	//M_EXECUTE VARIABLES //
		TP_READ						: LTP;  //Tempo de cadencement FB Modbus
		RTrig						: R_Trig; //Front montant sur TP_READ.Q
		ReadBusy					: BOOL;	//FB Modbus en busy



	
END_VAR

METHOD M_Execute
//////////////////
//  Method Calls 
/////////////////

VAR 
	// Method local variables (reinitialized at each cycle) 
	
	SppNum: UINT;
MesDataExd.MesData.NV: INT;
	SetTempSlope: REAL;
END_VAR

FOR KK_ModbusRead:=1 TO 2 DO
	AX_Error[KK_ModbusRead] 			:= Emul_MesModbusReadAlarm[KK_ModbusRead] ;
	
END_FOR

// INV 
SppNum:= SEL(ParamUnitID>11 ,1 , 2) ; 
		
			AX_PTR[SppNum].A1_INV_Smartlogger.Emul_RS(SET1:= IN_CmdStop, RESET:=IN_CmdStart ) ; 
			IF Emul_AlarmINV  THEN 
			MesDataExd.MesData.MesIDState :=16#0300 ;

			ELSIF AX_PTR[SppNum].A1_INV_Smartlogger.Emul_RS.Q1 THEN 
			MesDataExd.MesData.MesIDState:=16#0304 ;

			ELSIF MesP_INVmppt=0 THEN 
			MesDataExd.MesData.MesIDState:=16#A000 ;
	
			ELSIF IN_SetptPlimit < ParamPn THEN 
			MesDataExd.MesData.MesIDState:=16#0202 ;

			ELSIF AX_PTR[SppNum].A1_INV_Smartlogger.Emul_ComError THEN 
			MesDataExd.MesData.MesIDState:=16#B000 ;

			ELSE
			MesDataExd.MesData.MesIDState:=16#0200 ;

			END_IF	
	// Pas de pente dans les onduleurs . 		
//			Emul_Smooth(Setpoint:= AX_SPP[SppNum].A1_SmartLogger.SetptPlimit/AX_SPP[SppNum].A1_SmartLogger.ParamNbINV , Slope :=5,DeadBand:=2,Range:= ParamPnom,CycleTime:=CstCycleTime_G,InitialValue:=0, Reset:=(A1_HPP.CalState =9) OR Emul_AlarmINV OR NOT(AX_SPP[SppNum].A1_TGBT.MesDataExd.MesData.MesMainCB), OutValue=> SetTempSlope ) ;
			SetTempSlope :=SEL( MesDataExd.MesData.MesAlarmCom ,  AX_PTR[SppNum].A1_INV_Smartlogger.IN_SetptPlimit/AX_PTR[SppNum].A1_INV_Smartlogger.ParamNbINV , AX_PTR[SppNum].A1_INV_Smartlogger.ParamPnomINV )  ; 

		MesDataExd.MesData.MesP 			:=SEL((A1_PP.MesState =9) OR AX_PTR[SppNum].A1_INV_Smartlogger.Emul_AlarmINV OR NOT(AX_PTR[SppNum].A1_MainMVCB_PTR.MesDataExd.MesData.MesClosed) , MIN(SetTempSlope , MesP_INVmppt),  0)  ; 
		MesDataExd.MesData.MesQ 			:= AX_PTR[SppNum].A1_INV_Smartlogger.IN_SetptQlimit/AX_PTR[SppNum].A1_INV_Smartlogger.ParamNbINV  ; 
		MesDataExd.MesData.MesPdc 			:= MesDataExd.MesData.MesP/AX_PTR[SppNum].A1_INV_Smartlogger.MesDataExd.MesData.MesEff; 
		MesDataExd.MesData.MesIdc 			:= MesDataExd.MesData.MesPdc 	MesDataExd.MesData.MesUdc; 



MesDataExd.MesData.MesU 			:= AX_PTR[SppNum].A1_INV_Smartlogger.MesDataExd.MesData.MesU12 ; 
MesDataExd.MesData.MesV			    := MesDataExd.MesData.MesU/SQRT(3)*2 ; 
MesDataExd.MesData.MesI			    := SEL.MesDataExd.MesData.MesU = 0 , MesDataExd.MesData.MesP*1000 MesDataExd.MesData.MesU /SQRT(3) ,0 ) ; 
MesDataExd.MesData.MesFreq			:=  A1_SUBMV.A1_PM.MesDataExd.MesData.Mesfreq; 
MesDataExd.MesData.MesS			    := SQRT.MesDataExd.MesData.MesP.MesDataExd.MesData.MesP.MesDataExd.MesData.MesQ.MesDataExd.MesData.MesQ) ; 

MesDataExd.MesData.MesCosPhi			:=  0.95  ; 
MesDataExd.MesData.MesTemp			:= 32 ;  


// Other Variables
//MesDataExd.MesData.MesInsuResistor			:= 1220 ; 	

// Properties update. 
MesDataExd.MesData.MesAlarmCom	:= MesDataExd.MesData.MesIDState = 16#B000 ; 

//MesDataExd.MesData.MesAlm1		:= MesDataExd.MesData.MesIDState = 16#0300 ;
MesDataExd.MesData.ParamPn		:= 60  ; 

//MesDataExd.MesData.CalCurtailing	:= MesDataExd.MesData.MesStatus = 16#0201 OR MesDataExd.MesData.MesStatus = 16#0202; 
	

MesDataExd.MesData.MesUdc			:= 200 ;
MesDataExd.MesData.MesInsuResistor 	:= 150 ;
//MesDataExd.MesData.MesPF			:=0.97 ; 


//INV Exd
MesDataExd.MesEDay			:= 1000 ; 
MesDataExd.MesETot			:=  1100; 
MesDataExd.MesI1			:= MesDataExd.MesData.MesI; 
MesDataExd.MesI2			:= MesDataExd.MesData.MesI; 
MesDataExd.MesI3			:= MesDataExd.MesData.MesI; 
MesDataExd.MesU12			:=  AX_PTR[SppNum].A1_INV_Smartlogger.MesDataExd.MesData.MesU12; 
MesDataExd.MesU23			:=   AX_PTR[SppNum].A1_INV_Smartlogger.MesDataExd.MesData.MesU23; 
MesDataExd.MesU31			:=   AX_PTR[SppNum].A1_INV_Smartlogger.MesDataExd.MesData.MesU31; 
MesDataExd.MesV1			:= MesDataExd.MesData.MesV; 
MesDataExd.MesV2			:= MesDataExd.MesData.MesV;  
MesDataExd.MesV3			:= MesDataExd.MesData.MesV; 


// Properties update.
MesDataExd.MesData.MesI := MesDataExd.MesData.MesI1 + MesDataExd.MesData.MesI2 + MesDataExd.MesData.MesI3)/3;
MesDataExd.MesData.MesV := MesDataExd.MesData.MesV1 + MesDataExd.MesData.MesV2 + MesDataExd.MesData.MesV3)/3;
MesDataExd.MesData.MesS := SQRT.MesDataExd.MesData.MesP.MesDataExd.MesData.MesP + MesDataExd.MesData.MesQ.MesDataExd.MesData.MesQ);

MesDataExd.MesData.MesCurtl := MesDataExd.MesData.MesIDState=16#0202 OR MesDataExd.MesData.MesIDState=16#0203 ; 
//MesDataExd.MesData.ParamPnom := ParamPnom ;
END_METHOD

END_FUNCTION_BLOCK

// ---- 01_Equipement_Library/IPC/FB_IPC.TcPOU
FUNCTION_BLOCK FB_IPC

VAR_INPUT PERSISTENT 
	ParamTempoRestart		: TIME 	:= T#30S ;	(*  (s)Tempo to wait before resupplying the IPC*)
	
END_VAR
      	
VAR_INPUT           	
	Heure_Local     		: TIMESTRUCT;
	IN_CmdRestart 			: BOOL;	
	IN_CmdReset_L			: BOOL;			// (NA) External Reset Command
	
END_VAR     

VAR_OUTPUT
	//Child objects
	OUT_CmdOpen_IO			: BOOL;	
END_VAR        	
      	
VAR                 	
	bInit					: BOOL := TRUE;	// Booleen d'initialisation
		
	TP_Restart				: TP;
	// State Mananger //
	MesState				: BYTE; 		// Cal  : state
	
	// M_Evaluate //	
	MesData			: IPC;
	
END_VAR

METHOD M_Execute : BOOL
VAR_INPUT
END_VAR
END_METHOD

END_FUNCTION_BLOCK

// ---- 01_Equipement_Library/Operation Meter/FB_PM_520_230.TcPOU
FUNCTION_BLOCK FB_PM_520_230 EXTENDS FB_PM_Base
//////////////////
// Measurement Solution based on Digiware, but access through PMS Socomec
//////////////////
VAR CONSTANT
	// Characteristics of the object (Same for all instances)
			
END_VAR

VAR_INPUT PERSISTENT
	// Parameters of the Object (instance specific) 
	ParamUnitID					: BYTE 		:= 1 ;								// (NA)unit ID
	ParamInInterfaceSub			: BOOL := TRUE; // Serial interface RS422/RS485 TYPE (0:EL6021,1:SUB9)			
END_VAR

VAR_OUTPUT
	//Child objects
	
END_VAR
VAR
	//M_ALARMMANAGEMENT VARIABLES//
	                                                    								
                                                        								

	//M_READ VARIABLES//
		ModbusRTU					: FB_ModbusRTU;				// (NA) FB for Modbus Reading
				// (NA) Start address of the read
		//MesDataExd				: PM520;								// (NA) Structure of the PM3250
		
		ObjectCom					: INT;									// (NA) Sequence index
									
		Busy						: BOOL;
		StepRead					: UINT;									// (NA) Step for reading 2 blocks of registers
		AX_TrigRead					: ARRAY[1..1] OF R_trig;
		MbStruct					: ARRAY[1..1] OF Struct_InputRTU;	
		MesBlock					: ARRAY[1..1] OF ARRAY[1..120] OF WORD;	
		AX_Addr						: ARRAY[1..1] OF UINT 	:= [19000];
		AX_Qty						: ARRAY[1..1] OF UINT	:= [86];
		AX_UnitId					: ARRAY[1..1] OF BYTE	:= [1];
		AX_Function					: ARRAY[1..1] OF UINT	:= [4];	
		AX_Priority					: ARRAY[1..1] OF UINT	:= [1];
		KK							: INT;
		ComError 					: BOOL;
	//M_INIT VARIABLES //
		OutFBCompleteted			: BOOL;
	// M_EXECUTE VARIABLES //
		
                              

 
END_VAR

METHOD M_Execute
//////////////////
//  Method Calls 
/////////////////
VAR 

	
END_VAR
END_METHOD

END_FUNCTION_BLOCK

// ---- 01_Equipement_Library/Operation Meter/FB_PM_Base.TcPOU
FUNCTION_BLOCK FB_PM_Base 
//////////////////
// Measurement Solution. Base FB
//////////////////
VAR_INPUT PERSISTENT
	// Parameters of the Object (instance specific) 
	ParamTempoComAlarm			: TIME 			:= T#10S ; 						// (s) Config : Tempo to detect LOC Alarm
	ParamClockReadTime 			: TIME 			:= TIME#200MS;	  				// (ms) Read Modbus Frequency.  
	ParamTimeout				: TIME  		:= T#2S ;			  			// (s) Timeout for modbus reading
	
	
END_VAR

VAR_INPUT
	//Child objects
	IN_CmdToggleRead				: BOOL ; 
	IN_CmdReset_L					: BOOL ;	// (NA) External Reset Command

END_VAR
VAR
	//M_ALARMMANAGEMENT VARIABLES//
		TON_ComAlarm				: TON ; 												// Tempo before detecting loss of communication. 
	    TON_ComWarning				: TON ; 												// Tempo before detecting loss of one frame.                                               								
                                            								
												//(NA) [P,H] Communication Error with D50 Digiware (all chain ) 
		MesWarningCom				: BOOL ; 												// True if bad communication .

	//M_READ VARIABLES//
//	MesDataExd				AT %Q*: PM ; 
		ClockRead					AT %Q*: BOOL ; 												// Clock Read

	//M_INIT VARIABLES //
		bInit						: BOOL 				:= TRUE ; 							// (NA) Initialize object parameters at first cycle 
		
	// M_EXECUTE VARIABLES //
		TP1							: TP ; 												// (NA) Tempo to define Modbus Reading Frequency  
		
		//MesCP_Read					: BOOL;													// (NA) Permanent conditions to activate method
        Trig_Cmd_Read				: R_TRIG;                       
	// EMULATOR //                      
		
 
END_VAR

METHOD M_Execute
//////////////////
//  Method Calls 
/////////////////
VAR 
	// Method local variables (reinitialized at each cycle) 
	// EMULATOR

	
END_VAR
END_METHOD

END_FUNCTION_BLOCK

// ---- 01_Equipement_Library/Operation Meter/FB_PM_A40.TcPOU
FUNCTION_BLOCK FB_PM_A40 EXTENDS FB_PM_Base
//////////////////
// Measurement Solution based on Digiware, but access through PMS Socomec
//////////////////

VAR_INPUT PERSISTENT
	// Parameters of the Object (instance specific) 
	ParamUnitID					: BYTE := 22; 							// (NA) All unit ID For the Device (I35 + 1 U20)                                                                    			
	                                                                            			
	ParamIPAddress			   	: STRING := '192.168.20.15'; 								// (NA) IP Adress of D50 .
	ParamTCPPort				: UINT := 502;		// Modbus TCP Port


END_VAR

VAR_OUTPUT
	//Child objects
	
END_VAR
VAR
	//M_ALARMMANAGEMENT VARIABLES//
		
	//M_READ VARIABLES//
		FB_ModbusRead_I1			: ARRAY[1..2] OF  FB_ModbusRead ; 			// (NA) FB for Modbus Reading
	                                                                                    	
		MesBlock1_Temp 				: ARRAY[1..2] 	OF ARRAY[0..124] OF WORD;		//(NA) Temporary Block with multiple modbus reading (U30 + I35)
		MesModbusReadAlarm 		  	: ARRAY[1..2] OF BOOL ; 						// (NA) Modbus Read Alarm for communication 
		
		
		MesModbusAlarmCode			: ARRAY[1..2] OF UDINT;						// (NA) Modbus Read Alarm Code	
		
	//M_INIT VARIABLES //
		
	// M_EXECUTE VARIABLES //
		   	MesDataExd AT %Q*			: PM_Standard ;               


 
END_VAR

METHOD M_Execute
//////////////////
//  Method Calls 
/////////////////
VAR 
MesDataExd.MesData.dl 		: PDL_Exd;
	MesStateCB 		: BOOL;
MesDataExd.MesData.ull		: PM;
	
	KK: INT;
END_VAR
 MesDataExd.MesData.dl := A1_SUBMV.MesDataExd.MesData.

MesStateCB := A1_SUBMV.A1_MainMVCB.MesDataExd.MesData.MesClosed ; 
MesData.MesP := 0 ;
MesData.MesQ := 0 ; 


IF MesStateCB THEN
MesDataExd.MesData.MesU 	:= 230;
MesDataExd.MesData.MesU12 	:= 230;
MesDataExd.MesData.MesU23 	:= 230;
MesDataExd.MesData.MesU31 	:= 230;
MesDataExd.MesData.MesV 	:= A1_PP.MesDataExd.MesData.MesU/SQRT(3);
MesDataExd.MesData.MesV1 	:= A1_PP.MesDataExd.MesData.MesU/SQRT(3);
MesDataExd.MesData.MesV2 	:= A1_PP.MesDataExd.MesData.MesU/SQRT(3);
MesDataExd.MesData.MesV3 	:= A1_PP.MesDataExd.MesData.MesU/SQRT(3);
MesDataExd.MesData.MesFreq := A1_PP.MesDataExd.MesData.MesFreq;
	
	

MesDataExd.MesData.MesP 	:= 120  ;
MesDataExd.MesData.MesQ 	:= -20 ;
	
	
MesDataExd.MesData.MesP1 	:= MesDataExd.MesData.MesP ;
MesDataExd.MesData.MesP2 	:= 0 ;
MesDataExd.MesData.MesP3 	:= 0 ;

MesDataExd.MesData.MesQ1 	:= MesDataExd.MesData.MesQ;
MesDataExd.MesData.MesQ2 	:= 0;
MesDataExd.MesData.MesQ3 	:= 0;
MesDataExd.MesData.MesS := SQRT( MesDataExd.MesData.MesP * MesDataExd.MesData.MesP + MesDataExd.MesData.MesQ.MesDataExd.MesData.MesQ ) ; 
	
MesDataExd.MesData.MesI 	:= MesDataExd.MesData.MesS/(SQRT(3)*A1_PP.MesDataExd.MesData.MesU);
MesDataExd.MesData.MesI1 	:= MesDataExd.MesData.MesS/(SQRT(3)*A1_PP.MesDataExd.MesData.MesU);

ELSE 
MesDataExd.MesData.:= MesDataExd.MesData.ull;
END_IF

IF MesDataExd.MesData.MesP > 0 THEN
MesDataExd.MesData.MesE_AcDel := MesDataExd.MesData.MesE_AcDel + MesDataExd.MesData.MesP*ParamCycleTime_Emul/3600000	;
END_IF
IF MesDataExd.MesData.MesP < 0 THEN
MesDataExd.MesData.MesE_AcRec := MesDataExd.MesData.MesE_AcRec -.MesDataExd.MesData.MesP*ParamCycleTime_Emul/3600000	;
END_IF
IF MesDataExd.MesData.MesQ > 0 THEN
MesDataExd.MesData.MesE_ReacDel := MesDataExd.MesData.MesE_ReacDel + MesDataExd.MesData.MesQ*ParamCycleTime_Emul/3600000	;
END_IF
IF MesDataExd.MesData.MesQ < 0 THEN
MesDataExd.MesData.MesE_ReacRec := MesDataExd.MesData.MesE_ReacRec -.MesDataExd.MesData.MesQ*ParamCycleTime_Emul/3600000	;
END_IF

MesDataNull.MesE_ReacRec := MesDataExd.MesData.MesE_ReacRec;	
MesDataNull.MesE_ReacDel := MesDataExd.MesData.MesE_ReacDel;	
MesDataNull.MesE_AcRec := MesDataExd.MesData.MesE_AcRec;		
MesDataNull.MesE_AcDel := MesDataExd.MesData.MesE_AcDel;
END_METHOD

END_FUNCTION_BLOCK

// ---- 01_Equipement_Library/Operation Meter/FB_PM_ION7650.TcPOU
FUNCTION_BLOCK FB_PM_ION7650 EXTENDS FB_PM_Base
//////////////////
// Measurement Solution based on Digiware, but access through PMS Socomec
//////////////////
VAR CONSTANT
	// Characteristics of the object (Same for all instances)
			
END_VAR

VAR_INPUT PERSISTENT
	// Parameters of the Object (instance specific) 
	ParamUnitID					: BYTE 		:= 1 ;								// (NA)unit ID
//	ParamInInterfaceSub			: BOOL := TRUE; // Serial interface RS422/RS485 TYPE (0:EL6021,1:SUB9)
	ParamIPAdress		   		: STRING 	:= '192.168.20.15'; 				// (NA) IP Adress of ION7650 .
	ParamTcpPort				: UINT 		:= 502;					
	
END_VAR

VAR_OUTPUT
	//Child objects
	
END_VAR
VAR
	//M_ALARMMANAGEMENT VARIABLES//
	                                                    								                                          								

	//M_READ VARIABLES//
		FB_ModbusRead				: FB_ModbusRTU ;					// (NA) FB for Modbus Reading
		InputStructRead 			: ARRAY[1..1] OF  Struct_InputRTU;
		
		AX_Quantity					: ARRAY[1..1] OF WORD;					// (NA) Quantity of blocks to read
		AX_Address					: ARRAY[1..1] OF WORD;					// (NA) Start address of the read
		MesBlock_Temp 				: ARRAY[1..1] OF ARRAY[1..125] OF WORD;	// (NA) Temporary Block with multiple modbus reading (U30 + I35)
		Busy						: BOOL;
		OutErrorMbRead				: ARRAY[1..1] OF BOOL;
		
		RTrigI						: R_TRIG;
	//M_INIT VARIABLES //
		OutFBCompleteted			: BOOL;
	// M_EXECUTE VARIABLES //
 
	MesDataExd AT %Q*				: PM_Standard ;
END_VAR

METHOD M_Execute
//////////////////
//  Method Calls 
/////////////////
VAR 
	// Method local variables (reinitialized at each cycle) 
	// EMULATOR
		Psoltot		 : REAL;		// Total Solar Power 
		KK			 : BYTE;		// For Loop
	
		MesStateCB 	 : BOOL;
		MesDataNull 	: PM_Standard ;
		
	MesEReactCons_Temp: REAL;
	MesEActProd_Temp: REAL;
	MesEActCons_Temp: REAL;
	MesEReactProd_Temp: REAL;
END_VAR
MesStateCB 	 :=   A1_SUBMV.A1_MainMVCB.MesDataExd.MesData.MesClosed ; 
MesDataExd.MesData.MesP := - A1_SUBMV.A1_PM_Aux.MesDataExd.MesData.MesP ;	// initiliaze with auxiliaries power 
MesDataExd.MesData.MesQ := - A1_SUBMV.A1_PM_Aux.MesDataExd.MesData.MesQ   ; // aux + reactif in transfo  

IF MesStateCB THEN
MesDataExd.MesData.MesU 	:= A1_PP.MesData.MesU;
MesDataExd.MesData.MesU12 	:= A1_PP.MesData.MesU;
MesDataExd.MesData.MesU23 	:= A1_PP.MesData.MesU;
MesDataExd.MesData.MesU31 	:= A1_PP.MesData.MesU;
MesDataExd.MesData.MesV 	:= A1_PP.MesData.MesU/SQRT(3);
MesDataExd.MesData.MesV1 	:= A1_PP.MesData.MesU/SQRT(3);
MesDataExd.MesData.MesV2 	:= A1_PP.MesData.MesU/SQRT(3);
MesDataExd.MesData.MesV3 	:= A1_PP.MesData.MesU/SQRT(3);
MesDataExd.MesData.MesFreq := A1_PP.MesData.MesFreq;
	
	FOR KK:= 1 TO CstNbPTR_G DO 
	MesDataExd.MesData.MesP 	:= AX_PTR[KK].MesDataExd.MesData.MesP + MesDataExd.MesData.MesP;  //- ParamLossImpedance * SEL(AX_PTR[KK].MesDataExd.MesData.ProtectRelay_FLAIR.MesDataExd.MesData.MesU12 =0,  EXPT(((AX_PTR[KK].MesDataExd.MesData.MesP*1000) / AX_PTR[KK].MesDataExd.MesData.ProtectRelay_FLAIR.MesDataExd.MesData.MesU12/SQRT(3)),2) , 0 )/1000  ;		// Create some error due to transfo 
	MesDataExd.MesData.MesQ 	:= AX_PTR[KK].MesDataExd.MesData.MesQ + MesDataExd.MesData.MesQ ;
	END_FOR
	
MesDataExd.MesData.MesQ 	:= MesDataExd.MesData.MesQ + ABS(MesDataExd.MesData.MesP) * 0.1 	; // Add transfo conso
	
MesDataExd.MesData.MesP1 	:= MesDataExd.MesData.MesP ;
MesDataExd.MesData.MesP2 	:= MesDataExd.MesData.MesP ;
MesDataExd.MesData.MesP3 	:= MesDataExd.MesData.MesP ;

MesDataExd.MesData.MesQ1 	:= MesDataExd.MesData.MesQ;
MesDataExd.MesData.MesQ2 	:= MesDataExd.MesData.MesQ;
MesDataExd.MesData.MesQ3 	:= MesDataExd.MesData.MesQ;
MesDataExd.MesData.MesS := SQRT( MesDataExd.MesData.MesP * MesDataExd.MesData.MesP + MesDataExd.MesData.MesQ*MesDataExd.MesData.MesQ ) ; 
	
MesDataExd.MesData.MesI 	:= MesDataExd.MesData.MesS/(SQRT(3)*A1_PP.MesData.MesU);
MesDataExd.MesData.MesI1 	:= MesDataExd.MesData.MesS/(SQRT(3)*A1_PP.MesData.MesU);
MesDataExd.MesData.MesI2 	:= MesDataExd.MesData.MesS/(SQRT(3)*A1_PP.MesData.MesU);
MesDataExd.MesData.MesI3 	:= MesDataExd.MesData.MesS/(SQRT(3)*A1_PP.MesData.MesU);
ELSE 
	MesEActProd_Temp 	:= MesDataExd.MesData.MesEActProd 	 ;
	MesEActCons_Temp  := MesDataExd.MesData.MesEActCons   ;
	MesEReactProd_Temp:= MesDataExd.MesData.MesEReactProd ;
	MesEReactCons_Temp:= MesDataExd.MesData.MesEReactCons ;
	
//MesDataExd.MesData := MesDataNull;
MesDataExd.MesData.MesEActProd  	:=MesEActProd_Temp 	  ;
MesDataExd.MesData.MesEActCons  	:=MesEActCons_Temp    ;
MesDataExd.MesData.MesEReactProd	:=MesEReactProd_Temp  ;
MesDataExd.MesData.MesEReactCons	:=MesEReactCons_Temp  ;	
	
END_IF

IF MesDataExd.MesData.MesP > 0 THEN
MesDataExd.MesData.MesEActProd := MesDataExd.MesData.MesEActProd + MesDataExd.MesData.MesP*ParamCycleTime_Emul/3600000	;
END_IF
IF MesDataExd.MesData.MesP < 0 THEN
MesDataExd.MesData.MesEActCons := MesDataExd.MesData.MesEActCons - MesDataExd.MesData.MesP*ParamCycleTime_Emul/3600000	;
END_IF
IF MesDataExd.MesData.MesQ > 0 THEN
MesDataExd.MesData.MesEReactProd := MesDataExd.MesData.MesEReactProd + MesDataExd.MesData.MesQ*ParamCycleTime_Emul/3600000	;
END_IF
IF MesDataExd.MesData.MesQ < 0 THEN
MesDataExd.MesData.MesEReactCons := MesDataExd.MesData.MesEReactCons - MesDataExd.MesData.MesQ*ParamCycleTime_Emul/3600000	;
END_IF

MesDataNull.MesData.MesEReactCons := MesDataExd.MesData.MesEReactCons;	
MesDataNull.MesData.MesEReactProd := MesDataExd.MesData.MesEReactProd;	
MesDataNull.MesData.MesEActCons := MesDataExd.MesData.MesEActCons;		
MesDataNull.MesData.MesEActProd := MesDataExd.MesData.MesEActProd;
END_METHOD

END_FUNCTION_BLOCK

// ---- 01_Equipement_Library/Operation Meter/FB_PM_Janitza.TcPOU
FUNCTION_BLOCK FB_PM_Janitza EXTENDS FB_PM_Base
//////////////////
// Measurement Solution based on Janitza, but access through JemaPLC
//////////////////

VAR_INPUT PERSISTENT
	// Parameters of the Object (instance specific) 
	ParamIPAdress			   	: STRING 		:= '192.168.1.30'; 				// (NA) IP Adress of D50 .
	ParamUnitID 				: BYTE  := 1; 			  							// (NA)   Modbus Unit ID.	


END_VAR

VAR_OUTPUT
	//Child objects
	
END_VAR
VAR
	//M_ALARMMANAGEMENT VARIABLES//
	
	//M_READ VARIABLES//
		FB_ModbusRead_I1			: ARRAY[1..1] OF  FB_ModbusRead ; 		// (NA) FB for Modbus Reading
	
		MesBlock1_Temp 				: ARRAY[0..125] OF WORD;	//(NA) Temporary Block with multiple modbus reading (U30 + I35)
		
		MesModbusReadAlarm 		  	: ARRAY[1..1] OF BOOL ; 					// (NA) Modbus Read Alarm for communication 
		
		MesModbusAlarmCode			: UDINT;												// (NA) Modbus Read Alarm Code	
		
	//M_INIT VARIABLES //

	// M_EXECUTE VARIABLES //
			MesDataExd AT %Q*				: PM_Standard ;
	
END_VAR

METHOD M_Execute
//////////////////
//  Method Calls 
/////////////////
VAR 
	// Method local variables (reinitialized at each cycle) 
	// EMULATOR
	// Method local variables (reinitialized at each cycle) 
	///MesDataExd.MesData.dl 		: SUBMV_Exd;
	MesStateCB 		: BOOL;
MesDataExd.MesData.ull		: PM;
	
	KK: INT;
	
END_VAR
//MesDataExd.MesData.dl	 := A1_SUBMV.MesDataExd.MesData.

MesStateCB 	 := A1_SUBMV.A1_MainMVCB.MesDataExd.MesData.MesClosed ; 
MesData.MesP := - A1_SUBMV.A1_PM_Aux.MesDataExd.MesData.MesP ;	// initiliaze with auxiliaries power 
MesData.MesQ := - A1_SUBMV.A1_PM_Aux.MesDataExd.MesData.MesQ   ; // aux + reactif in transfo  


IF MesStateCB THEN
MesDataExd.MesData.MesU 	:= A1_PP.MesDataExd.MesData.MesU;
MesDataExd.MesData.MesU12 	:= A1_PP.MesDataExd.MesData.MesU;
MesDataExd.MesData.MesU23 	:= A1_PP.MesDataExd.MesData.MesU;
MesDataExd.MesData.MesU31 	:= A1_PP.MesDataExd.MesData.MesU;
MesDataExd.MesData.MesV 	:= A1_PP.MesDataExd.MesData.MesU/SQRT(3);
MesDataExd.MesData.MesV1 	:= A1_PP.MesDataExd.MesData.MesU/SQRT(3);
MesDataExd.MesData.MesV2 	:= A1_PP.MesDataExd.MesData.MesU/SQRT(3);
MesDataExd.MesData.MesV3 	:= A1_PP.MesDataExd.MesData.MesU/SQRT(3);
MesDataExd.MesData.MesFreq := A1_PP.MesDataExd.MesData.MesFreq;
	
	
	FOR KK:= 1 TO CstNbESS_G DO 
		//MesDataExd.MesData.MesP 	:= AX_PTR[KK].MesDataExd.MesData.MesP + MesDataExd.MesData.MesP  - ParamLossImpedance * SEL(AX_PTR[KK].MesDataExd.MesData.MesU=0,  EXPT(((AX_PTR[KK].MesDataExd.MesData.MesP*1000) / AX_PTR[KK].MesDataExd.MesData.MesU/SQRT(3)),2) , 0 )/1000  ;		// Create some error due to transfo 
	MesDataExd.MesData.MesQ 	:= AX_PTR[KK].MesDataExd.MesData.MesQ + MesDataExd.MesData.MesQ ;
	END_FOR
	
	
MesDataExd.MesData.MesQ 	:= MesDataExd.MesData.MesQ + ABS(MesDataExd.MesData.MesP) * 0.1 	; // Add transfo conso
	
	
MesDataExd.MesData.MesP1 	:= MesDataExd.MesData.MesP ;
MesDataExd.MesData.MesP2 	:= MesDataExd.MesData.MesP ;
MesDataExd.MesData.MesP3 	:= MesDataExd.MesData.MesP ;

MesDataExd.MesData.MesQ1 	:= MesDataExd.MesData.MesQ;
MesDataExd.MesData.MesQ2 	:= MesDataExd.MesData.MesQ;
MesDataExd.MesData.MesQ3 	:= MesDataExd.MesData.MesQ;
MesDataExd.MesData.MesS := SQRT( MesDataExd.MesData.MesP * MesDataExd.MesData.MesP + MesDataExd.MesData.MesQ.MesDataExd.MesData.MesQ ) ; 
	
MesDataExd.MesData.MesI 	:= MesDataExd.MesData.MesS/(SQRT(3)*A1_PP.MesDataExd.MesData.MesU);
MesDataExd.MesData.MesI1 	:= MesDataExd.MesData.MesS/(SQRT(3)*A1_PP.MesDataExd.MesData.MesU);
MesDataExd.MesData.MesI2 	:= MesDataExd.MesData.MesS/(SQRT(3)*A1_PP.MesDataExd.MesData.MesU);
MesDataExd.MesData.MesI3 	:= MesDataExd.MesData.MesS/(SQRT(3)*A1_PP.MesDataExd.MesData.MesU);
ELSE 
MesDataExd.MesData.:= MesDataExd.MesData.ull;
END_IF

IF MesDataExd.MesData.MesP > 0 THEN
MesDataExd.MesData.MesEActProd := MesDataExd.MesData.MesEActProd + MesDataExd.MesData.MesP*ParamCycleTime_Emul/3600000	;
END_IF
IF MesDataExd.MesData.MesP < 0 THEN
MesDataExd.MesData.MesEActCons := MesDataExd.MesData.MesEActCons -.MesDataExd.MesData.MesP*ParamCycleTime_Emul/3600000	;
END_IF
IF MesDataExd.MesData.MesQ > 0 THEN
MesDataExd.MesData.MesEReactProd := MesDataExd.MesData.MesEReactProd + MesDataExd.MesData.MesQ*ParamCycleTime_Emul/3600000	;
END_IF
IF MesDataExd.MesData.MesQ < 0 THEN
MesDataExd.MesData.MesEReactCons := MesDataExd.MesData.MesEReactCons -.MesDataExd.MesData.MesQ*ParamCycleTime_Emul/3600000	;
END_IF

MesDataNull.MesEReactCons := MesDataExd.MesData.MesEReactCons;	
MesDataNull.MesEReactProd := MesDataExd.MesData.MesEReactProd;	
MesDataNull.MesEActCons := MesDataExd.MesData.MesEActCons;		
MesDataNull.MesEActProd := MesDataExd.MesData.MesEActProd;
END_METHOD

END_FUNCTION_BLOCK

// ---- 01_Equipement_Library/Operation Meter/FB_PM_PM3250.TcPOU
FUNCTION_BLOCK FB_PM_PM3250 EXTENDS FB_PM_Base
//////////////////
// Measurement Solution based on Digiware, but access through PMS Socomec
//////////////////
VAR CONSTANT
	// Characteristics of the object (Same for all instances)
			
END_VAR

VAR_INPUT PERSISTENT
	// Parameters of the Object (instance specific) 
	ParamUnitID					: BYTE 		:= 1 ;								// (NA)unit ID
//	ParamInInterfaceSub			: BOOL := TRUE; // Serial interface RS422/RS485 TYPE (0:EL6021,1:SUB9)			
END_VAR

VAR_OUTPUT
	//Child objects
	
END_VAR
VAR
	//M_ALARMMANAGEMENT VARIABLES//

	//M_READ VARIABLES//

		InputStructRead 			: ARRAY[1..5] OF  Struct_InputRTU;

		AX_Quantity					: ARRAY[1..5] OF WORD;					// (NA) Quantity of blocks to read
		AX_Address					: ARRAY[1..5] OF WORD;					// (NA) Start address of the read
		MesBlock_Temp 				: ARRAY[1..5] OF ARRAY[1..125] OF WORD;	// (NA) Temporary Block with multiple modbus reading (U30 + I35)
		Busy						: BOOL;
		OutErrorMbRead				: ARRAY[1..5] OF BOOL;
	

	//M_INIT VARIABLES //
		OutFBCompleteted			: BOOL;
	// M_EXECUTE VARIABLES //
		RTrigI						: R_TRIG;
		MesDataExd		AT %Q*			: PM_Standard ;

 
END_VAR

METHOD M_Execute
//////////////////
//  Method Calls 
/////////////////
VAR 
	// Method local variables (reinitialized at each cycle) 
	// EMULATOR
		Psoltot			: REAL;		// Total Solar Power  
		KK				: BYTE;		// For Loop
		MesDataNull		: PM;
		MesStateCB      : BOOL;
		
	 	

END_VAR

	

MesStateCB := A1_SUBMV.A1_MainMVCB.MesDataExd.MesData.MesClosed AND A1_SUBMV.A1_GridMVCB.MesDataExd.MesData.MesClosed AND A1_SUBMV.A1_AuxMVCB.MesDataExd.MesData.MesClosed ; 
MesDataExd.MesData.MesP := 0 ;
MesDataExd.MesData.MesQ := 0 ; 


IF MesStateCB THEN
	MesDataExd.MesData.MesU 	:= 230;
	MesDataExd.MesData.MesU12 	:= 230;
	MesDataExd.MesData.MesU23 	:= 230;
	MesDataExd.MesData.MesU31 	:= 230;
	MesDataExd.MesData.MesV 	:= A1_PP.MesData.MesU/SQRT(3);
	MesDataExd.MesData.MesV1 	:= A1_PP.MesData.MesU/SQRT(3);
	MesDataExd.MesData.MesV2 	:= A1_PP.MesData.MesU/SQRT(3);
	MesDataExd.MesData.MesV3 	:= A1_PP.MesData.MesU/SQRT(3);
	MesDataExd.MesData.MesFreq := A1_PP.MesData.MesFreq;
	
	

	MesDataExd.MesData.MesP 	:= 120  ;
	MesDataExd.MesData.MesQ 	:= -20 ;
	
	
	MesDataExd.MesData.MesP1 	:= MesDataExd.MesData.MesP ;
	MesDataExd.MesData.MesP2 	:= 0 ;
	MesDataExd.MesData.MesP3 	:= 0 ;

	MesDataExd.MesData.MesQ1 	:= MesDataExd.MesData.MesQ;
	MesDataExd.MesData.MesQ2 	:= 0;
	MesDataExd.MesData.MesQ3 	:= 0;
	MesDataExd.MesData.MesS := SQRT( MesDataExd.MesData.MesP *  MesDataExd.MesData.MesP + MesDataExd.MesData.MesQ*MesDataExd.MesData.MesQ ) ; 
	
	MesDataExd.MesData.MesI 	:= MesDataExd.MesData.MesS/(SQRT(3)* A1_PP.MesData.MesU);
	MesDataExd.MesData.MesI1 	:= MesDataExd.MesData.MesS/(SQRT(3)* A1_PP.MesData.MesU);

	IF MesDataExd.MesData.MesP > 0 THEN
		MesDataExd.MesData.MesEActProd := MesDataExd.MesData.MesEActProd  + MesDataExd.MesData.MesP*ParamCycleTime_Emul/3600000	;
	END_IF
	IF MesDataExd.MesData.MesP < 0 THEN
		MesDataExd.MesData.MesEActCons :=  MesDataExd.MesData.MesEActCons - MesDataExd.MesData.MesP*ParamCycleTime_Emul/3600000	;
	END_IF
	IF MesDataExd.MesData.MesQ > 0 THEN
		MesDataExd.MesData.MesEReactProd := MesDataExd.MesData.MesEReactCons + MesDataExd.MesData.MesQ*ParamCycleTime_Emul/3600000	;
	END_IF
	IF MesDataExd.MesData.MesQ < 0 THEN
		MesDataExd.MesData.MesEReactCons :=  MesDataExd.MesData.MesEReactCons - MesDataExd.MesData.MesQ*ParamCycleTime_Emul/3600000	;
	END_IF
	
	
	
END_IF
END_METHOD

END_FUNCTION_BLOCK

// ---- 01_Equipement_Library/Operation Meter/FB_PM_PM800.TcPOU
FUNCTION_BLOCK FB_PM_PM800 EXTENDS FB_PM_Base
VAR_INPUT
		IPAddrAI 	: STRING;	// Adresse IP Requête Analogic Inputs
END_VAR
VAR_OUTPUT
END_VAR
VAR
MesDataExd AT %Q*	: PM_PM800 ;
	
	// Modbus Read Variables
	FB_ModbusReadAI : ARRAY[1..2] OF FB_ModbusRead ;
	
	// Temp Blocks Filled by Requests
	AI_List_1 	    : ARRAY[1..128] OF WORD ;
	AI_List_2 		: ARRAY[1..128] OF WORD ;
	
	tTimeout 		: TIME := T#2S ;
	
END_VAR

METHOD M_AlarmManagement
VAR_INPUT
END_VAR
//////////////////
// Digiware measurement tool alarm and warning management
/////////////////

VAR 
	// Method local variables (reinitialized at each cycle) 
	FB_AlarmCodeManager			: FB_AlarmCodeManager ; 
	
	ComWarning					: BOOL;			// Error in one of the Modbus Requests
	ComAlarm					: BOOL;			// Error in both Modbus Requests
	
END_VAR
ComWarning 	:= FB_ModbusReadAI[1].ModbusReadAlarm OR FB_ModbusReadAI[2].ModbusReadAlarm;
ComAlarm 	:= FB_ModbusReadAI[1].ModbusReadAlarm AND FB_ModbusReadAI[2].ModbusReadAlarm;
	
TON_ComAlarm(IN:= ComAlarm , PT:= ParamTempoComAlarm, Q= MesDataExd.MesData.MesAlarmCom) ;	
TON_ComWarning(IN:= ComWarning  , PT:= ParamTempoComAlarm, Q=>MesWarningCom) ;	

//					General com alarm : All the read FB fucked up


// ALARM CODE //
	FB_AlarmCodeManager(
		bAlarm1			:= MesDataExd.MesData.MesAlarmCom  , 					// Communication Alarm #COM
		bAlarm2			:=FALSE, // 
		bAlarm3			:=FALSE, // 
		bAlarm4			:=FALSE, // 
		bAlarm5			:=FALSE, //
		bAlarm6			:=FALSE, //
		bAlarm7			:=FALSE, //
		bAlarm8			:=FALSE, //
		bAlarm9			:=FALSE, //
		bAlarm10		:=FALSE, //
		bAlarm11		:=FALSE, //
		bAlarm12		:=FALSE, //
		bAlarm13		:=FALSE, //
		bAlarm14		:=FALSE, //
		bAlarm15		:= FALSE , 			// 			 
		wAlarmCode		=>MesDataExd.MesData.MesAlarmCode);

// WARNING CODE //
	FB_AlarmCodeManager(		
		bAlarm1			:=MesWarningCom	,				 // Communication Warning #COM
		bAlarm2			:=FALSE, 		// 
		bAlarm3			:=FALSE, 		// 
		bAlarm4			:=FALSE, 		// 
		bAlarm5			:=FALSE, //
		bAlarm6			:=FALSE, //
		bAlarm7			:=FALSE, //
		bAlarm8			:=FALSE, //
		bAlarm9			:=FALSE, //
		bAlarm10		:=FALSE, //
		bAlarm11		:=FALSE, //
		bAlarm12		:=FALSE, //
		bAlarm13		:=FALSE, //
		bAlarm14		:=FALSE, //
		bAlarm15		:=FALSE, //
		wAlarmCode		=>MesDataExd.MesData.MesWarningCode);		

// EVENT CODE //
END_METHOD

END_FUNCTION_BLOCK

// ---- 01_Equipement_Library/Operation Meter/FB_PM_SicamQ100.TcPOU
FUNCTION_BLOCK FB_PM_SicamQ100 EXTENDS FB_PM_Base
VAR_INPUT
		ParamIPAddress				: STRING 	:= '192.168.20.66'; 	// (NA)Config: IP Adress of PV INverter
		ParamUnitID 				: BYTE  	:= 1; 			  		// (NA)   Modbus Unit ID. 
		ParamTCPPort				: UINT		:= 502;					// (NA) TCP port for modbus

END_VAR
VAR_OUTPUT
END_VAR
VAR
	// M_READ VARIABLES//

	MesDataExd			: PM_SicamQ100 ; 
		AX_STR						: ARRAY [1..CstNbSB_INV_G] OF STR;
		AX_ModbusRead		   		: ARRAY [1..3] OF FB_ModbusRead ; 					// (NA) FB for Modbus Reading
		
		MesBlock1_Temp 				: ARRAY[1..2]  OF WORD; 			// (NA) Temporary Block with multiple modbus reading (Caution : Double Word variables)
		MesBlock2_Temp 				: ARRAY[1..76]  OF WORD; 			// (NA) Temporary Block with multiple modbus reading (Caution : Double Word variables)
		MesBlock3_Temp 				: ARRAY[1..38]  OF WORD; 			// (NA) Temporary Block with multiple modbus reading (Caution : Double Word variables)

		AX_ReadAlarm 		  		: ARRAY [1..3] OF BOOL ; 							// (NA) Modbus Read Alarm for all modbus frames		
		AX_ReadAlarmCode			: ARRAY [1..3] OF UDINT;							// (NA) Modbus Read Alarm Code		
		AX_ReadBusy					: ARRAY [1..3] OF BOOL;								// (NA) Modbus Read Busy  
		AX_ReadCompleted			: ARRAY [1..3] OF BOOL;								// (NA) Modbus Read Completed
				
	// M_STATEMANAGER//
		bErrorState					: BOOL;								//(NA) Inverter is in incoherent state
		
		
	

END_VAR

END_FUNCTION_BLOCK

// ---- 01_Equipement_Library/Operation Meter/FB_PM_SM103E.TcPOU
FUNCTION_BLOCK FB_PM_SM103E EXTENDS FB_PM_Base
//////////////////
// Measurement Solution based on Digiware, but access through PMS Socomec
//////////////////
VAR CONSTANT
	// Characteristics of the object (Same for all instances)
			
END_VAR

VAR_INPUT PERSISTENT
	// Parameters of the Object (instance specific) 
	ParamUnitID					: BYTE 		:= 5 ;								// (NA)unit ID
	

END_VAR

VAR_OUTPUT
	//Child objects
	
END_VAR
VAR
	//M_ALARMMANAGEMENT VARIABLES//	                                                    							                                                								

	//M_READ VARIABLES//

	bReadError					: BOOL;
	bReadCompleted 				: BOOL;
	bReadBusy					: BOOL;
	InputStructRead 			: Struct_InputRTU;



	bReadError2					: BOOL;
	bReadCompleted2 				: BOOL;
	bReadBusy2					: BOOL;
	InputStructRead2 			: Struct_InputRTU;
	
	MesBlock1_Temp 				: ARRAY[1..64]  OF WORD; 		// (NA) Temporary Block with multiple mod
	MesBlock2_Temp 				: ARRAY[1..20]  OF WORD; 		// (NA) Temporary Block with multiple mod

		
		
	//M_INIT VARIABLES //
	
	// M_EXECUTE VARIABLES //
		RTrigI						: R_TRIG;

	MesDataExd AT %Q*			: PM_Standard ;


 
END_VAR

END_FUNCTION_BLOCK

// ---- 01_Equipement_Library/PCS/FB_PCS_Base.TcPOU
FUNCTION_BLOCK FB_PCS_Base
//////////////////
// PCS controller . Base FB
//////////////////

VAR_INPUT PERSISTENT
	// Parameters of the Object (instance specific) 
	ParamUnitID 					: BYTE  	:= 1; 			  		// (NA)   CTRLPcs Modbus Unit ID.
	ParamIPAddress			   		: STRING 	:= '192.168.1.64'; 		// (NA) Config IP Adress of CTRLPCs
	ParamTcpPort					: UINT		:= 502;
	ParamNbPcs						: BYTE	 	:= 3 ; 					// (NA) Config : Number of Pcs/Module controlled . 
                                                                
	ParamTempoComAlarm				: TIME 		:= T#10S ; 				// (s) Config : Tempo to detect LOC Alarm
	ParamTempoComWarning			: TIME 		:= T#5S ; 				// (s) Config : Tempo to detect LOC Alarm
//	ParamTimeOutBlckStrt			: TIME 		:= T#3M ;				// (s) Config : Tempo to start before Timeout warning

	ParamClockReadTime 				: TIME 		:= TIME#200MS;	  		// (ms) Read Modbus Frequency .   
	ParamClockWriteTime 			: TIME 		:= TIME#500MS;   		// (ms) Write Modbus Frequency .         
	ParamTimeout					: TIME  	:= T#4S ;		  		// (s) Timeout for modbus reading                                                              	
	ParamTimePulseTrig				: TIME 		:= T#4S;            	// (s)
	                                                                	
	ParamEssNum						: UINT 		:= 1;					// (NA) ID number of the Pcs' father PCS
	ParamPcsNum						: UINT 		:= 1;					// (NA) ID number of the PCS 
END_VAR

VAR_OUTPUT
	//Child objects
	
END_VAR

VAR_INPUT
	// I/O Inputs 
		// ALARM MANAGEMENT //
		IN_SetptP					: REAL ;						// (kW)   [P,H] Dynamic aCtive Power  setpoint 
		IN_SetptQ					: REAL ;						// (kVAr) [P,H] Dynamic reactive Power setpoint 
		IN_SetptU					: REAL ;						// (kW)   [P,H] Dynamic aCtive Power  setpoint 
		IN_SetptF					: REAL ;						// (kW)   [P,H] Dynamic aCtive Power  setpoint 
		IN_SetptCosPhi				: REAL;							// (NA)  [P,H] Dynamic CosPhi setpoint	
		IN_CmdReset					: BOOL ;
		IN_CmdToggleRead			: BOOL;
        IN_CmdToggleWrite			: BOOL;
		
		
	
END_VAR

VAR
	//M_ALARMMANAGEMENT VARIABLES//
		TON_ComAlarm				: TON ; 			// Tempo before deteting loss of communication. 
		TON_ComWarning				: TON ; 			// Tempo before deteting loss of communication. 
		
                                         
		CmdResetPcs					: BOOL ; 			// (NA) [P,H] 	Reset alarms and warning
		MesWarningCom				: BOOL ; 			// (NA) [P,H]   True if bad communication 
		MesAlarmCom					: BOOL ; 			// (NA) True if complete loss of modbus communication 

	//M_CP VARIABLES//
		Trig_Cmd_Read				: R_TRIG;                                                                                        
		Trig_Cmd_Write				: R_TRIG;                                                                                        
        
        
		
	//M_WRITECOMMAND VARIABLES//
	
		CmdStart					: BOOL;							// (NA) [P,H] External Start Command
		CmdStop 					: BOOL; 						// (NA) [P,H] External Stop CommAND   

	//M_STATEMANAGER VARIABLES//
		MesState					: BYTE ; 						// (NA) Cal [P,H,B] Bit0: 1 = Not Available (AC or DC breaker open or AllAcContactorsOpened), Bit1: GridMode: 1=grid	
	
	//M_WRITESETPOINTS VARIABLES//
	
		FB_CheckSetpt1				: FB_CheckSetpt ; 				// (NA) Functionnal Block to check if active power Writing Successful
		FB_CheckSetpt2				: FB_CheckSetpt ; 				// (NA) Functionnal Block to check if reactive power Writing Successful

	//M_INIT VARIABLES //
		bInit						: BOOL 			:= TRUE ; 		// (NA) Initialize object parameters at first cycle 
		
	// M_EXECUTE VARIABLES //
		TP1							: TP ; 						// (NA) Tempo to define Modbus Reading Frequency 
		TP2 						: TP ; 						// (NA) Tempo to define Modbus Writing Frequency
                                    
		ClockRead		AT%Q*		: BOOL;							// (NA) Modbus reading Clock
		TrigRead 					: R_TRIG;							// (NA) Modbus writing Clock 	
		ClockWrite 		AT%Q*		: BOOL;							// (NA) Modbus writing Clock 	
		TrigWrite 					: R_TRIG;							// (NA) Modbus writing Clock 	
		CalCP_Start                 : BOOL ; 						// (NA) Permanent conditions to activate method
		CalCP_Stop                  : BOOL ;                       	// (NA) Permanent conditions to activate method   	
	    CalCP_Reset                 : BOOL ; 						// (NA) Permanent conditions to activate method  
		MesCP_Read					: BOOL := TRUE;	(* Read function enable *)
		MesCP_Write					: BOOL := TRUE;	(* Write function enable *)	
		
		
END_VAR

METHOD M_Evaluate : BOOL
VAR_INPUT
END_VAR
END_METHOD

METHOD M_Execute
//////////////////
//  Method Calls 
/////////////////

VAR 
	// Method local variables (reinitialized at each cycle) 
	KK			: BYTE;			// For Loop 
	
END_VAR


// METHODS CALLS //
	IF bInit THEN
		M_Init() ; 
		bInit					:= FALSE ; 
	ELSIF CmdInit_G THEN 
		bInit:= TRUE ;
		
	END_IF

	M_Read() ; 
	M_Evaluate();                                                               
	M_WriteCommand() ; 
	
// COM MANAGER //
END_METHOD

METHOD M_Init

VAR 

END_VAR
END_METHOD

METHOD M_Read
//////////////////
//  Read Modbus Variable for PCS . 
/////////////////

VAR 
	// Method local variables (reinitialized at each cycle) 


END_VAR
END_METHOD

METHOD M_WriteCommand
//////////////////
//  Modbus Write of the command for the PCS. 
/////////////////

VAR 
	// Method local variables (reinitialized at each cycle) 


END_VAR
END_METHOD

END_FUNCTION_BLOCK

// ---- 01_Equipement_Library/PCS/FB_PCS_Jema.TcPOU
FUNCTION_BLOCK FB_PCS_Jema EXTENDS FB_PCS_Base
//////////////////
// PLC controller. Jema Object 
//////////////////
VAR_INPUT 
	MesGridForming						: BOOL;

	ParamFvP_Droop						: REAL := 0.02; // P(F) = a x F + b, a = ParamFvP_Droop
	ParamUvQ_Droop						: REAL := 0.02;
          
	FB_RampP							: FB_Ramp ; 
	FB_RampQ							: FB_Ramp ; 
        
	MesPInitial							: REAL;
	MesQInitial							: REAL;
	Trig_ClockRead						: R_TRIG;
	Trig_ClockWrite						: ARRAY[1..3] OF  R_TRIG;
	CmdWrite							: ARRAY[1..3] OF BOOL;
	AX_Cmd				AT%Q*			: ARRAY[1..3] OF ARRAY [1..120] OF WORD;
	AX_Cmd_New							: ARRAY[1..3] OF ARRAY [1..120] OF WORD;
	bTest								: BOOL;
END_VAR
VAR_INPUT PERSISTENT
	// Parameters of the Object
		ParamPrange							: REAL := 1559.0 ; // (kW) Power range for sMesIng . 
		ParamPn							: REAL := 1300.0;	// (kW) Nominal power
		ParamQn							: REAL := 1300.0;	// (kW) Nominal power
		
		ParamIPAddress_DSP					: ARRAY[1..3] OF  STRING ; 	

    	                            		
		ParamSetPtModbusMode				: BOOL:= TRUE;		// If True, then Setpoints come from Modbus
		ParamPoverQ							: BOOL:= TRUE;		// If P over Q is True, then Max setpoint for Q calculated from setpoint of P
    	                    			
		ParamQfU_UDbHigh    				: REAL;				// (V)JEMA U1 : AKUO U_UDbHigh
		ParamQfU_Umax		    			: REAL;				// (V)JEMA U2 : AKUO U_Umax
		ParamQfU_UDbLow	    				: REAL;				// (V)JEMA U3 : AKUO U_UDbLow
		ParamQfU_Umin		    			: REAL;				// (V)JEMA U4 : AKUO U_Umin
		                            		
		ParamQfU_QDbHigh					: REAL;				// (kVAr)JEMA Q1 : AKUO U_QDbHigh. Power per power column (between -500 and 500)
		ParamQfU_Qmax						: REAL;				// (kVAr)JEMA Q4 : AKUO U_Qmax. Power per power column (between -500 and 500)
		ParamQfU_QDbLow						: REAL;				// (kVAr)JEMA Q3 : AKUO U_QDbLow. Power per power column (between -500 and 500)
		ParamQfU_Qmin						: REAL;				// (kVAr)JEMA Q2 : AKUO U_Qmin. Power per power column (between -500 and 500)
    	                            		
		ParamPfF_FDbHigh	    			: REAL;				// (Hz)JEMA f1 : AKUO P_FDbHigh
		ParamPfF_Fmax		    			: REAL;				// (Hz)JEMA f2 : AKUO P_Fmax
		ParamPfF_FDbLow	    				: REAL;				// (Hz)JEMA f3 : AKUO P_FDbLow
		ParamPfF_Fmin		    			: REAL;				// (Hz)JEMA f4 : AKUO P_Fmin
		                            		
		ParamPfF_PDbHigh					: REAL;				// (kW) JEMA P1 : AKUO P_PDbHigh	 Power per power column
		ParamPfF_Pmax						: REAL;				// (kW)JEMA P2 : AKUO P_Pmax. Power per power column
		ParamPfF_PDbLow						: REAL;				// (kW)JEMA P3 : AKUO P_PDbLow. Power per power column
		ParamPfF_Pmin						: REAL;				// (kW)JEMA P4 : AKUO P_Pmin. Power per power column
    	
		ParamPfF_FhystLow					: REAL;				// (Hz)JEMA fst1
		ParamPfF_FhystHigh					: REAL;				// (Hz)JEMA fst2
 

		ParamClockWriteTimeFreqReg			: TIME := T#3S ; 
   	         	    		
		ParamTimeSoCRangeReachedRmp			: TIME;				// (ms) Time to ramp P back to the setpoint after the SoC reached its limits
		ParamTimeFreqRegStbDuration			: TIME;				// (ms) Time to wait after entering the stable before ramping the P back to the setpoint 
		ParamTimeStblRmp					: TIME; 			// (ms) Time to ramp P back to the setpoint after entering the stable 
		    
 
	ParamTempoStandby				: TIME	:= T#10S;	// (s)Tempo to let time for PCS to apply a 0 setpoint before stopping . 

   	                           
   	
		ParamFreqRegSoCmax 					: REAL;	 			// (%) Jema Stops charging setpoint and overfreq regulation if BESS reaches this value
		ParamFreqRegSoCmin 					: REAL;				//(%) Jema Stops discharging setpoint and underfreq regulation if BESS reaches this value
    	
		ParamLVRT_Enabled					: BOOL; 			// LVRT Enabled 
		ParamAntiIslanding_Enabled			: BOOL:=TRUE;				// Is Anti Islanding enabled

		ParamDeactivateWatchdog				: BOOL:=TRUE;				// Parameter to deactivate the watchdog

	// Not Used at the moment : used to calculate theoretical Efficiency
		ParamRendementPcsNom				: REAL := 98;		// (%) Nominal Efficiency of the PCS at optimal conditions  
		ParamRendementPcsMin				: REAL := 80;		// (%) Minimal Efficiency of the PCS at P = 0  
		ParamTauxDeChargeRef				: REAL := 10;		// (%) LoadFactor where 1/5 of the efficiency is reached  

	// 
		ParamTimeoutCmdQ					: TIME := T#15S; 	// (s) Time to activate or deactivate Q regulation before an alarm is raised
		ParamTimeoutCmdCosPhi				: TIME := T#15S; 	//  (s)Time to activate or deactivate CosPhi regulation before an alarm is raised
		ParamTimeoutQvU						: TIME := T#15S;	//  (s)Time to activate or deactivate Q(U) regulation before an alarm is raised
		ParamTimeoutPvF						: TIME := T#15S;	// (s) Time to activate or deactivate P(f) regulation before an alarm is raised
 		ParamTimeoutGridFeederTransition	: TIME := T#1M;		// (min) Time elapsed after grid feeder cmd when an alarm is raised   
 		ParamTimeoutOffTransition			: TIME := T#1M;		// (min) Time elapsed after CmdStop cmd when an alarm is raised
 
           			
END_VAR 
VAR_INPUT   	                   			
	// Commands :
		IN_CmdPcsInLocalMode				: BOOL;				// PCS is not included in available PCS' pool (excluded from PP control). 
		IN_CmdStopOperation					: BOOL;				// BESS Specific command : Stop operation		
		IN_CmdPreventStart					: BOOL;				// BESS Specific command : Prevent start	
		IN_CmdOpenAC						: BOOL;				// Cmd To send an Open AC order
		IN_CmdOpenDC						: BOOL;				// Cmd To send an Open DC order	
 		IN_CmdP_On							: BOOL:=TRUE;				// Cmd start regulating on SetptP from outside of PCS : if you wan to know from what source, add a _IO2 value
		IN_CmdQ_On							: BOOL;				// Cmd start regulating on SetptQ from outside of PCS : if you wan to know from what source, add a _IO2 value
		IN_CmdCosPhi_On						: BOOL;				// Cmd start regulating on SetptCosPhi from outside of PCS : if you wan to know from what source, add a _IO2 value
		IN_CmdP_Off							: BOOL;				// Cmd start regulating on SetptP from outside of PCS : if you wan to know from what source, add a _IO2 value
		IN_CmdQ_Off							: BOOL;				// Cmd start regulating on SetptQ from outside of PCS : if you wan to know from what source, add a _IO2 value
		IN_CmdCosPhi_Off					: BOOL;				// Cmd start regulating on SetptCosPhi from outside of PCS : if you wan to know from what source, add a _IO2 value
		IN_CmdFreqregOn						: BOOL;				// Cmd 
		IN_CmdFreqregOff					: BOOL;				// 
		IN_CmdUregOn						: BOOL;				// 
		IN_CmdUregOff						: BOOL;				// 

		
		IN_CmdStandby						: BOOL;				// Cmd To send a soft Stop (No opening and closing of the AC/DC switch \m/ )
		IN_CmdStart							: BOOL;				// Cmd To send a start to the PCS (Does the full procedure, Soft + Close AC + Close DC)
		IN_CmdStop							: BOOL;				// Cmd To send a stop to the PCS (Soft Stop + Open DC + Open AC)
		                            		

		IN_CmdGridFeeder					: BOOL;				// 
		IN_SetptP_Local						: REAL;				// Local Command
		IN_SetptQ_Local						: REAL;				// Local Command
		
		IN_CmdWatchdog						: BOOL ; 			// Activate or Deactivate the Watchdog function

                
END_VAR
VAR_OUTPUT
	//Child objects
		OUt_SetptP_IO					: INT;			// (NA) Analogical value for the active power setpoint (based on ParamPn)
		OUT_SetptQ_IO					: INT;			// (NA) Analogical value for the reactive power setpoint (based on ParamQn)

END_VAR
VAR                                     	
	//M_ALARMMANAGEMENT VARIABLES//     	
	//M_READ VARIABLES//            		
		ModbusRead            				: ARRAY [1..CstNbPowerCol_PCS_G+1] OF FB_ModbusRead ; 	// (NA) FB for Modbus Reading
		MesBlock1_Temp						: ARRAY [1..CstNbPowerCol_PCS_G+1] OF ARRAY[1..120] OF WORD ; // (NA) Temporary Block Matrix for PCS modbus reading		
		AX_PcsHeartbit						: ARRAY [1..CstNbPowerCol_PCS_G] OF BOOL;
		                                	
	///MesDataExd.MesData.cs_Jema						: ARRAY [1..CstNbModule_Pcs] OF PCSJema ; 			// (NA) [H,B] PCS  Data Structure
		MesModbusReadAlarm 		  			: ARRAY [1..CstNbPowerCol_PCS_G+1] OF BOOL ;				// (NA) Modbus Read Alarm for communication
		TON_PcsHeartBitAlarm				: ARRAY [1..CstNbPowerCol_PCS_G] OF TON ;	
		TON_AlarmPcs						: ARRAY [1..CstNbPowerCol_PCS_G] OF TON ; 		// DesInhibate undervoltage alarms on PCS few seconds after PCS connected .  
                                        	
		DFV									: ARRAY[1..3] OF FB_DetectFixedValue;	
		StaticValuesToCompareHeartbit		: ARRAY[1..3] OF REAL;
		                                	                                     
		CTU_PcsNb							: CTU ; 
	
	// M_EVALUATE VARIABLES//
//		DataPP								: PP;
//		DataSUB_MV								: SUB_MV_Exd;
		DataSystemBMS						: SystemBMS;
		MesWatchdog					: BOOL;
		MesHeartbeat_Old					: WORD;
		Trig_Watchdog						: R_TRIG;
		CalNbFreqActivePcs					: UINT;			// Number of powercolumn that have frequency regulation 
		RS_hystlimitmin						: RS;
		RS_hystlimitmax						: RS;
                            		
	//M_WRITECOMMAND VARIABLES//    		
		ModbusWrite							: ARRAY [1..5] OF FB_ModbusWrite ;		// (NA) Functionnal Block for Writing Command Word through modbus
		Trig_Write							: ARRAY [1..5] OF R_TRIG;
		MesModbusWriteCmdAlarm				: ARRAY [1..5] OF BOOL ;				// (NA) Modbus Write Failed  (Command word) . 	
		MesModbusWriteCode          		: ARRAY [1..5] OF UDINT ; 				// (NA) Modbus Write Alarm Code 
		CmdWrite			AT%Q*			: ARRAY [1..5] OF BOOL;
		AX_Cmd				AT%Q*			: ARRAY [1..5] OF ARRAY [1..120] OF WORD;
		AX_Cmd_Old							: ARRAY [1..5] OF ARRAY [1..120] OF WORD;
                                   		
		TRIG_CmdOpenAC						: R_TRIG;			// Trig to detect an order to change Mode
		TRIG_CmdOpenDC						: R_TRIG;			// Trig to detect an order to change Mode
		TRIG_CmdP_On						: R_TRIG;			// Trig to detect an order to change Mode
		TRIG_CmdQ_On			    		: R_TRIG;			// Trig to detect an order to change Mode
		TRIG_CmdCosPhi_On 					: R_TRIG;			// Trig to detect an order to change Mode
		TRIG_CmdP_Off						: R_TRIG;			// Trig to detect an order to change Mode
		TRIG_CmdQ_Off			    		: R_TRIG;			// Trig to detect an order to change Mode
		TRIG_CmdCosPhi_Off 					: R_TRIG;			// Trig to detect an order to change Mode
		TRIG_CmdReset						: R_TRIG;		
		TRIG_FreqReg_On						: R_TRIG;
		TRIG_FreqReg_Off					: R_TRIG;
		TRIG_UReg_On						: R_TRIG;
		TRIG_UReg_Off						: R_TRIG;
	
		
		TOF_FreqRegDisable					: TOF;			// Inhibe frequency regulation when frequency is zero  
		R_TRIG_FreqRegDisable				: R_TRIG;		// Reactivate after a few seconds to initiaize
		
		
		
		
		
		TRIG_CmdGridFeeder					: R_TRIG;
	
		TRIG_CmdStop						: R_TRIG;
		TRIG_CmdStandby						: R_TRIG;
		TRIG_CmdStart						: R_TRIG;
	
	F_TRIG_Standby: F_TRIG;		                            		

		TP_Reset							: TP ; 				// (NA) Maintain Reset command for a certain time 
		TP_CmdStandby						: TP;				// TP To maintain a soft stop order
		TP_CmdStandbyDelay					: TP ; 				// TP to delay application of standby order
		
		
		
		bMaintainStop					: BOOL;	// Allow to keep setpoint to zero after a standby order .   RS .     	

		FB_Ramp_Standby			: FB_Ramp;	// Ramp to zero after a standby order
		FB_Ramp_StandbyQ		: FB_Ramp; // Ramp to zero after a standby order
	
		

		// Pour la commande start, j'envoie une consigne pour fermer les contacteurs DC des batteries
		TP_CmdOpenAC						: TP;				// TP To ensure R trig is detected
		TP_CmdOpenDC						: TP;				// TP To ensure R trig is detected

		TP_CmdStart							: TP;				// TP To ensure R trig is detected
		TP_CmdPreStart						: TP;				// TP To send a close dc breaker order before sending start order
		F_TrigPreStart						: F_TRIG;			// failing edge to detect end of TP;
		
		// Pour la commande stop, pour éviter qu'on ouvre tout d'un coup, je faire un pré stop pendant 1,5s où j'envoie un autre de standby
		TP_CmdStop							: TP;				// TP To ensure R trig is detected
		TP_CmdPreStop						: TP;				// TP to send a soft stop before sending a stop 
		F_TrigPreStop						: F_TRIG;			// failing edge to detect end of TP;
		                            		
		TON_CmdP_On							: TON;			// Detect the non execution of an order
		TON_CmdQ_On			    			: TON;			// Detect the non execution of an order
		TON_CmdCosPhi_On 					: TON;			// Detect the non execution of an order
		TON_CmdP_Off						: TON;			// Detect the non execution of an order
		TON_CmdQ_Off			    		: TON;			// Detect the non execution of an order
		TON_CmdCosPhi_Off 					: TON;			// Detect the non execution of an order
		TON_FreqReg_On						: TON;
		TON_FreqReg_Off						: TON;
		TON_UReg_On							: TON;
		TON_UReg_Off						: TON;
		TON_CmdGridFeeder					: TON;
		TON_CmdStart			    		: TON;
		TON_CmdStop	                		: TON;
		TON_CmdStandby		        		: TON;

		    
		TP3					: TP ; // For freq reg Clockwrite
		TrigWriteFreqReg	: R_TRIG ; 
		ClockWriteFreqReg	: BOOL ; 
                        		
END_VAR

METHOD M_Evaluate : BOOL
VAR_INPUT
END_VAR
VAR
	MesDataExd.MesData.DL 		: PDL_Exd;
MesDataExd.MesData.bms 	: SystemBMS;
	KK				: INT;
	
	MesS 			: ARRAY[1..3] OF REAL;
	MesS2 			: REAL;
	MesS3 			: REAL;
	NbPcsConnected 	: UINT;
	III				: INT;
	CBChoose		: BOOL ;


END_VAR
// Evaluate to get the values of the Storage + Substation
MesDataPDL 		:= A1_SUBMV.MesDataExd.MesData.
MesDataSbms 	:= AX_ESS[ParamEssNum].AX_Bbms[ParamPcsNum].MesDataExd.MesData.

// Mes frequence 
CASE ParamEssNum OF 
	1:
			CBChoose := A1_SUBMV.A1_CB_ImBess1.MesDataExd.MesData.MesClosed ; 
	2:
			CBChoose := A1_SUBMV.A1_CB_ImBess2.MesDataExd.MesData.MesClosed ; 
	3:
			CBChoose := A1_SUBMV.A1_CB_ImBess3.MesDataExd.MesData.MesClosed ; 
	4:
			CBChoose := A1_SUBMV.A1_CB_ImBess4.MesDataExd.MesData.MesClosed ; 
	5:
			CBChoose := A1_SUBMV.A1_CB_ImBess5.MesDataExd.MesData.MesClosed ; 
	6:
			CBChoose := A1_SUBMV.A1_CB_ImBess6.MesDataExd.MesData.MesClosed ; 

END_CASE

IF CBChoose THEN
	MesVacPcs 		:= MesDataExd.MesData.DL.AX_PM1.MesV / MesUGen*500;
	MesFreqPcs 		:= MesDataExd.MesData.DL.AX_PM1.MesFreq;
ELSE 
	MesVacPcs 		:= 0;	
    MesFreqPcs 		:= 0;
	CmdStop 		:= TRUE;
END_IF

MesUsetptWrittenScada	:= WORD_TO_REAL(AX_Cmd[1][15]);
MesUMesWrittenScada		:= WORD_TO_REAL(AX_Cmd[1][16]);

// Reset 
TON_Watchdog(In := AX_Cmd[1][38].0, PT := T#10S);
IF AX_Cmd[1][38].1 THEN
	FOR KK:= 1 TO ParamNbPcs DO 
	MesDataExd.MesData.AX_PCS[KK].MesJemaAlarms := Alarms_Null;
	END_FOR
END_IF

MesGridForming := AX_Cmd[1][38].2;

TRIG_CmdStart(CLK := AX_Cmd[1][38].5  OR SEL( ParamPcsNum=2, AX_ESS[ParamEssNum].OUT_CmdStartPcs1_IO ,AX_ESS[ParamEssNum].OUT_CmdStartPcs2_IO ) );
TRIG_CmdStop(CLK := AX_Cmd[1][38].6 OR CmdStop  OR AX_ESS[ParamEssNum].OUT_CmdEmergencyStop );
TRIG_CmdFreqReg(CLK := AX_Cmd[1][38].8);
TRIG_CmdUReg(CLK := AX_Cmd[1][38].9);	
TRIG_CmdStandby(CLK := AX_Cmd[1][38].15 OR SEL( ParamPcsNum=2, AX_ESS[ParamEssNum].OUT_CmdStopPcs1_IO ,AX_ESS[ParamEssNum].OUT_CmdStopPcs2_IO ) OR NOT CBChoose);	

MesSoCWrittenScada			:= WORD_TO_REAL(AX_Cmd[1][4]);
ParamFreqRegSoCmax			:= WORD_TO_REAL(AX_Cmd[1][2]);
ParamFreqRegSoCmin			:= WORD_TO_REAL(AX_Cmd[1][3]);



MesData.MesOnGrid := NOT AX_Cmd[1][38].2;
MesData.MesOffGrid := AX_Cmd[1][38].2;




// CmdStart
	IF TRIG_CmdStart.Q THEN
		MesSoftStop	:= FALSE;
	MesDataExd.MesData.MesAcBreaker := TRUE;
	END_IF
	TP_Precharge(IN := TRIG_CmdStart.Q AND NOT MesDataExd.MesData.MesDcBreaker, PT := T#3S);
MesDataExd.MesData.MesPrecharge := TP_Precharge.Q;
	FOR KK:= 1 TO ParamNbPcs DO 
	MesDataExd.MesData.AX_PCS[KK].MesUdc := MesDataExd.MesData.bms.MesUdc*TIME_TO_REAL(TP_Precharge.ET)/3000;
	END_FOR
	
	TRIG_PrechargeDone(CLK := TP_Precharge.Q);
	IF TRIG_PrechargeDone.Q THEN
	MesDataExd.MesData.MesDcBreaker := TRUE;
	END_IF

// Cmd Stop 
	IF TRIG_CmdStop.Q THEN
		CmdStop			:= FALSE;
	MesDataExd.MesData.MesAcBreaker := FALSE;
	MesDataExd.MesData.MesDcBreaker := FALSE;
		FOR KK := 1 TO ParamNbPcs DO
		MesDataExd.MesData.AX_PCS[KK].MesAcSwitchClosed := FALSE;
			//MesDataExd.MesData.MesOnGrid := FALSE;
			//MesDataExd.MesData.MesOffGrid := FALSE;
		END_FOR
	END_IF
// Cmd Soft Stop 
	IF TRIG_CmdStandby.Q  THEN
		MesSoftStop := TRUE;
		FOR KK := 1 TO ParamNbPcs DO
		MesDataExd.MesData.AX_PCS[KK].MesAcSwitchClosed := FALSE;
			//MesDataExd.MesData.MesOnGrid := FALSE;
			//MesDataExd.MesData.MesOffGrid := FALSE;
		END_FOR
	END_IF	
	
	MesVacPcs_Min := ParamQfU_Umin*500/MesUGen/SQRT(3);
	MesVacPcs_Max := ParamQfU_Umax*500/MesUGen/SQRT(3);
	
	FOR KK:= 1 TO ParamNbPcs DO 
		TP_CloseAcContact[KK](IN := MesDataExd.MesData.MesDcBreaker AND MesDataExd.MesData.MesAcBreaker AND MesVacPcs > MesVacPcs_Min AND MesVacPcs < MesVacPcs_Max AND NOT MesSoftStop, PT := T#5S);
		TRIG_CmdAcContact[KK](CLK := TP_CloseAcContact[KK].Q);
		IF TRIG_CmdAcContact[KK].Q THEN

		MesDataExd.MesData.AX_PCS[KK].MesAcSwitchClosed := TRUE;
		END_IF
	END_FOR
	
// Gestion de la puissance 
IF MesDataExd.MesData.MesDcBreaker THEN
	FOR KK := 1 TO ParamNbPcs DO
	MesDataExd.MesData.AX_PCS[KK].MesUdc	 		:= MesDataExd.MesData.bms.MesUdc;
	END_FOR
ELSE 
	FOR KK := 1 TO ParamNbPcs DO
	MesDataExd.MesData.AX_PCS[KK].MesUdc	 		:= 0;
	END_FOR
END_IF

// SoC Limit 
	TP_FreqRampToZeroSoClimit(IN := MesSoCWrittenScada > ParamFreqRegSoCmax OR MesSoCWrittenScada < ParamFreqRegSoCmin, PT := ParamTimeSoCRangeReachedRmp);
	TRIG_BeginRamp(CLK := TP_FreqRampToZeroSoClimit.Q);
	
	IF TRIG_BeginRamp.Q THEN
		MesPmaxRampSoClimit :=0 ; 
		FOR KK:= 1 TO ParamNbPcs DO 
			MesPmaxRampSoClimit := MesPmaxRampSoClimit + MesDataExd.MesData.AX_PCS[KK].MesPac ;
		END_FOR
	END_IF


// MesData
	FOR KK := 1 TO ParamNbPcs DO 
	MesDataExd.MesData.AX_PCS[KK].MesUac 	:= MesVacPcs*SQRT(3);
	MesDataExd.MesData.AX_PCS[KK].MesFreq 	:= MesFreqPcs;
		IF MesDataExd.MesData.AX_PCS[KK].MesAcSwitchClosed AND MesDataExd.MesData.AX_PCS[KK].MesUdc >0 AND MesDataExd.MesData.AX_PCS[KK].MesUac >0 THEN
			IF MesSoCWrittenScada > ParamFreqRegSoCmax AND MesDataExd.MesData.OUT_SetptP < 0 THEN
			MesDataExd.MesData.AX_PCS[KK].MesPac := (TIME_TO_REAL(TP_FreqRampToZeroSoClimit.PT) - TIME_TO_REAL(TP_FreqRampToZeroSoClimit.ET))/TIME_TO_REAL(TP_FreqRampToZeroSoClimit.PT) * MesPmaxRampSoClimit/ParamNbPcs; 
			ELSIF MesSoCWrittenScada < ParamFreqRegSoCmin AND MesDataExd.MesData.OUT_SetptP > 0 THEN
			MesDataExd.MesData.AX_PCS[KK].MesPac := (TIME_TO_REAL(TP_FreqRampToZeroSoClimit.PT) - TIME_TO_REAL(TP_FreqRampToZeroSoClimit.ET))/TIME_TO_REAL(TP_FreqRampToZeroSoClimit.PT) * MesPmaxRampSoClimit/ParamNbPcs; 
			ELSE
			MesDataExd.MesData.AX_PCS[KK].MesPac 	:= MesDataExd.MesData.AX_PCS[KK].MesPac+ MesDataExd.MesData.OUT_SetptP/ParamNbPcs -.MesDataExd.MesData.AX_PCS[KK].MesPac)/CoeffSuiviSetpointPcs ;
			END_IF
		MesDataExd.MesData.AX_PCS[KK].MesQac 	:= MesDataExd.MesData.AX_PCS[KK].MesQac+ MesDataExd.MesData.OUT_SetptQ/ParamNbPcs -.MesDataExd.MesData.AX_PCS[KK].MesQac)/CoeffSuiviSetpointPcs ;

			MesS[KK] 					:= SQRT( MesDataExd.MesData.AX_PCS[KK].MesPac.MesDataExd.MesData.AX_PCS[KK].MesPac.MesDataExd.MesData.AX_PCS[KK].MesQac.MesDataExd.MesData.AX_PCS[KK].MesQac));

		MesDataExd.MesData.AX_PCS[KK].MesPdc 	:= SEL.MesDataExd.MesData.AX_PCS[KK].MesPac < 0, MesDataExd.MesData.AX_PCS[KK].MesPac/0.96, MesDataExd.MesData.AX_PCS[KK].MesPac*0.96);	
		MesDataExd.MesData.AX_PCS[KK].MesI1 	:= MesS[KK]*1000/(SQRT(3).MesDataExd.MesData.AX_PCS[KK].MesUac);
		MesDataExd.MesData.AX_PCS[KK].MesI2 	:= MesDataExd.MesData.AX_PCS[KK].MesI1;
		MesDataExd.MesData.AX_PCS[KK].MesI3 	:= MesDataExd.MesData.AX_PCS[KK].MesI1;
		MesDataExd.MesData.AX_PCS[KK].MesIac 	:= MesDataExd.MesData.AX_PCS[KK].MesI1;
		MesDataExd.MesData.AX_PCS[KK].MesIdc 	:= MesDataExd.MesData.AX_PCS[kk].MesPdc *1000 //MesDataExd.MesData.AX_PCS[KK].MesUdc ;
		ELSE
		MesDataExd.MesData.AX_PCS[KK].MesPac 	:= 0;
		MesDataExd.MesData.AX_PCS[KK].MesQac 	:= 0;
		MesDataExd.MesData.AX_PCS[KK].MesI1  	:= 0;
		MesDataExd.MesData.AX_PCS[KK].MesI2  	:= 0;
		MesDataExd.MesData.AX_PCS[KK].MesI3  	:= 0;
		MesDataExd.MesData.AX_PCS[KK].MesIac 	:= 0;
		MesDataExd.MesData.AX_PCS[KK].MesIdc 	:= 0;
		MesDataExd.MesData.AX_PCS[KK].MesPdc 	:= 0;

		END_IF
	END_FOR


	FOR KK := 1 TO ParamNbPcs DO
		
	MesDataExd.MesData.AX_PCS[KK].MesTempCabinet 	:= 30.MesDataExd.MesData.AX_PCS[KK].MesPac/519*5;
	MesDataExd.MesData.AX_PCS[KK].MesTempControl 	:= 27.5.MesDataExd.MesData.AX_PCS[KK].MesPac/519*5;
	MesDataExd.MesData.AX_PCS[KK].MesTempPowerUnit := 32.5.MesDataExd.MesData.AX_PCS[KK].MesPac/519*5;
		NbPcsConnected := NbPcsConnected + SEL.MesDataExd.MesData.AX_PCS[1].MesAcSwitchClosed, 0, 1);
	END_FOR
MesDataExd.MesData.MesPnom := 1559.0/3.0*ParamNbPcs;
	
MesDataExd.MesData.MesAvailability := UINT_TO_REAL(NbPcsConnected) /ParamNbPcs*100.0;		// A mettre a zero si alarme ? 



// Regulation de fréquence
		RS_FreqIsAbove(SET := MesSoCWrittenScada < ParamFreqRegSoCmax AND MesFreqPcs > ParamPfF_FDbHigh, RESET1 := TRIG_FreqRampIsFinished.Q OR NOT MesDataExd.MesData.OUT_CmdFreqregMode	OR NOT CBChoose OR NbPcsConnected=0);	
		RS_FreqIsBelow(SET := MesSoCWrittenScada > ParamFreqRegSoCmin AND MesFreqPcs < ParamPfF_FDbLow, RESET1 := TRIG_FreqRampIsFinished.Q OR NOT MesDataExd.MesData.OUT_CmdFreqregMode	OR NOT CBChoose OR NbPcsConnected=0);	
		
	IF MesDataExd.MesData.OUT_CmdFreqregMode AND CBChoose THEN

		TON_FreqWaitInStableBeforeRamp
		(
			IN := (RS_FreqIsAbove.Q1 OR RS_FreqIsBelow.Q1) AND  MesFreqPcs > ParamPfF_FhystLow AND MesFreqPcs < ParamPfF_FhystHigh,
			PT := ParamTimeEnterStblPriorRmp
		);
			
		IF RS_FreqIsAbove.Q1 THEN
			FreqMaxForHyst := min(MAX(FreqMaxForHyst, MesFreqPcs), ParamPfF_Fmax);
			//PmaxForHyst := MAX((FreqMaxForHyst-ParamPfF_FDbHigh)/(ParamPfF_Fmax-ParamPfF_FDbHigh)*ParamPfF_Pmin, ParamPfF_Pmin);
		ELSIF RS_FreqIsBelow.Q1 THEN
			FreqMaxForHyst := MAX( MIN(FreqmaxForHyst, MesFreqPcs), ParamPfF_Fmin);
			//PmaxForHyst := MIN((FreqMaxForHyst-ParamPfF_FDbLow)/(ParamPfF_Fmin-ParamPfF_FDbLow)*ParamPfF_Pmax, ParamPfF_Pmax);
		ELSE
			FreqMaxForHyst := 50;
			PmaxForHyst := 0;
			MesPInitial	:= MesDataExd.MesData.AX_PCS[1].MesPac + MesDataExd.MesData.AX_PCS[2].MesPac + SEL( ParamNbPcs =3  ,0  , MesDataExd.MesData.AX_PCS[3].MesPac) ; //  MesDataExd.MesData.OUT_SetptP ; 
		END_IF
		
	
		TP_FreqRampToZeroOnceStable(IN := TON_FreqWaitInStableBeforeRamp.Q, pt := ParamTimeFreqRegStbDuration);
		TRIG_FreqRampIsFinished(CLK := TP_FreqRampToZeroOnceStable.Q);
		FB_RampP(IN:= MesPInitial/ParamNbPcs , ASCEND := ParamPnomPcs , DESCEND := ParamPnomPcs , TIMEBASE := ParamTimeFreqRegStbDuration, RESET:= FALSE ) ; 
		
		
		IF TRIG_FreqRampIsFinished.Q THEN
			FreqMaxForHyst := 50;
			PmaxForHyst := 0;
		END_IF
		FOR KK:= 1 TO ParamNbPcs DO 
			IF RS_FreqIsAbove.Q1 THEN
				IF ABS(ParamPfF_FDbHigh - ParamPfF_Fmax ) > 0.001 THEN 
				MesDataExd.MesData.AX_PCS[KK].MesPac := ( MesPInitial  + MAX((ParamPfF_Pmin *(ParamPfF_FDbHigh -FreqMaxForHyst ) - ParamPfF_PDbHigh*(ParamPfF_Fmax-FreqMaxForHyst) ) * 1/(ParamPfF_FDbHigh-ParamPfF_Fmax),  ParamPfF_Pmin)) /ParamNbPcs ;
				ELSE
				MesDataExd.MesData.AX_PCS[KK].MesPac := (MesPInitial + ParamPfF_Pmin) /ParamNbPcs ;
				
				END_IF
				IF TP_FreqRampToZeroOnceStable.Q THEN
					
				MesDataExd.MesData.AX_PCS[KK].MesPac :=FB_RampP.OUT ; // MesPInitial/ParamNbPcs + (TIME_TO_REAL(TP_FreqRampToZeroOnceStable.PT)-TIME_TO_REAL(TP_FreqRampToZeroOnceStable.ET))/TIME_TO_REAL(TP_FreqRampToZeroOnceStable.PT)*PmaxForHyst;

				ELSE
					FB_RampP(RESET:= TRUE , IN_RESET_VALUE := MesDataExd.MesData.AX_PCS[KK].MesPac) ; 
				END_IF
			END_IF
			IF RS_FreqIsBelow.Q1 THEN
				IF ABS(ParamPfF_Fmin - ParamPfF_FDbLow ) > 0.001 THEN 
				MesDataExd.MesData.AX_PCS[KK].MesPac := (MesPInitial + MIN(   ((ParamPfF_PDbLow - ParamPfF_Pmax)/(ParamPfF_FDbLow - ParamPfF_Fmin))*( FreqMaxForHyst - ParamPfF_FDbLow ) + ParamPfF_PDbLow ,  ParamPfF_Pmax) )/ParamNbPcs ;
				ELSE
				MesDataExd.MesData.AX_PCS[KK].MesPac := (MesPInitial+ ParamPfF_Pmax)/ParamNbPcs  ;
				END_IF
				IF TP_FreqRampToZeroOnceStable.Q THEN
					
				MesDataExd.MesData.AX_PCS[KK].MesPac :=FB_RampP.OUT ; // MesPInitial/ParamNbPcs+ (TIME_TO_REAL(TP_FreqRampToZeroOnceStable.PT) - TIME_TO_REAL(TP_FreqRampToZeroOnceStable.ET))/TIME_TO_REAL(TP_FreqRampToZeroOnceStable.PT)*PmaxForHyst;
				ELSE
					FB_RampP(RESET:= TRUE , IN_RESET_VALUE := MesDataExd.MesData.AX_PCS[KK].MesPac) ;
				END_IF
			END_IF
		END_FOR
	ELSE 
		FreqMaxForHyst := 50;
		PmaxForHyst := 0;
		MesPInitial	:= MesDataExd.MesData.AX_PCS[1].MesPac + MesDataExd.MesData.AX_PCS[2].MesPac + SEL( ParamNbPcs =3  ,0  , MesDataExd.MesData.AX_PCS[3].MesPac) ; ///MesDataExd.MesData.OUT_SetptP ; 
	END_IF

// Regulation de tension
		RS_VoltIsAbove(SET := MesUMesWrittenScada > ParamQfU_UDbHigh, RESET1 := TRIG_VoltRampIsFinished.Q OR NOT MesDataExd.MesData.OUT_CmdUregMode	OR NOT CBChoose OR NbPcsConnected=0);	
		RS_VoltIsBelow(SET := MesUMesWrittenScada < ParamQfU_UDbLow, RESET1 := TRIG_VoltRampIsFinished.Q OR NOT MesDataExd.MesData.OUT_CmdUregMode	OR NOT CBChoose OR NbPcsConnected=0);	
		
	IF MesDataExd.MesData.OUT_CmdUregMode AND CBChoose THEN

		TON_VoltWaitInStableBeforeRamp
		(
			IN := (RS_VoltIsAbove.Q1 OR RS_VoltIsBelow.Q1) AND  MesUMesWrittenScada > ParamQfU_UDbLow AND MesUMesWrittenScada < ParamQfU_UDbHigh,
			PT := ParamTimeEnterStblPriorRmp
		);
			
		IF RS_VoltIsAbove.Q1 THEN
			VoltMaxForHyst := min(MAX(VoltMaxForHyst, MesUMesWrittenScada), ParamQfU_Umax);
			//QmaxForHyst := MAX((VoltMaxForHyst-ParamQfU_UDbHigh)/(ParamQfU_Umax-ParamQfU_UDbHigh)*ParamQfU_Qmin, ParamQfU_Qmin);
		ELSIF RS_VoltIsBelow.Q1 THEN
			VoltMaxForHyst := MAX( MIN(VoltmaxForHyst, MesUMesWrittenScada), ParamQfU_Umin);
			//QmaxForHyst := MIN((VoltmaxForHyst-ParamQfU_UDbLow)/(ParamQfU_Umin-ParamQfU_UDbLow)*ParamQfU_Qmax, ParamQfU_Qmax);
		ELSE
			VoltMaxForHyst := 10000;
			QmaxForHyst := 0;
			MesQInitial	:= MesDataExd.MesData.OUT_SetptQ ; 
		END_IF
	
		TP_VoltRampToZeroOnceStable(IN := TON_VoltWaitInStableBeforeRamp.Q, pt := ParamTimeFreqRegStbDuration);
		TRIG_VoltRampIsFinished(CLK := TP_VoltRampToZeroOnceStable.Q);
		FB_RampQ(IN:= MesQInitial/ParamNbPcs , ASCEND := ParamPnomPcs , DESCEND := ParamPnomPcs , TIMEBASE := ParamTimeFreqRegStbDuration, RESET:= FALSE ) ; 

		IF TRIG_VoltRampIsFinished.Q THEN
			VoltMaxForHyst := 10000;
			QmaxForHyst := 0;
		END_IF
		
		FOR KK:= 1 TO ParamNbPcs DO 
			IF RS_VoltIsAbove.Q1 THEN
			MesDataExd.MesData.AX_PCS[KK].MesQac := MAX(MesQInitial/ParamNbPcs + (VoltMaxForHyst-ParamqfU_UDbHigh)/(ParamQfU_Umax-ParamqfU_UDbHigh)*ParamQfU_Qmin/ParamNbPcs, MesQInitial/ParamNbPcs + ParamQfU_Qmin/ParamNbPcs);
				IF TP_VoltRampToZeroOnceStable.Q THEN
				MesDataExd.MesData.AX_PCS[KK].MesQac := FB_RampQ.OUT ; //  MesQInitial/ParamNbPcs + (TIME_TO_REAL(TP_VoltRampToZeroOnceStable.PT)-TIME_TO_REAL(TP_VoltRampToZeroOnceStable.ET))/TIME_TO_REAL(TP_VoltRampToZeroOnceStable.PT)*QmaxForHyst/ParamNbPcs;
				ELSE
					FB_RampQ(RESET:= TRUE , IN_RESET_VALUE := MesDataExd.MesData.AX_PCS[KK].MesQac) ;
				END_IF
			END_IF
			IF RS_VoltIsBelow.Q1 THEN
			MesDataExd.MesData.AX_PCS[KK].MesQac := MIN(MesQInitial/ParamNbPcs + (VoltMaxForHyst-ParamQfU_UDbLow)/(ParamQfU_Umin-ParamQfU_UDbLow)*ParamQfU_Qmax/ParamNbPcs, MesQInitial/ParamNbPcs + ParamQfU_Qmax/ParamNbPcs);
			IF TP_VoltRampToZeroOnceStable.Q THEN
			MesDataExd.MesData.AX_PCS[KK].MesQac := FB_RampQ.OUT ; // MesQInitial/ParamNbPcs + (TIME_TO_REAL(TP_VoltRampToZeroOnceStable.PT) - TIME_TO_REAL(TP_VoltRampToZeroOnceStable.ET))/TIME_TO_REAL(TP_VoltRampToZeroOnceStable.PT)*QmaxForHyst/ParamNbPcs;
			ELSE
				FB_RampQ(RESET:= TRUE , IN_RESET_VALUE := MesDataExd.MesData.AX_PCS[KK].MesQac) ;
			END_IF
			END_IF
		END_FOR
	ELSE 
		VoltMaxForHyst := 10000;
		QmaxForHyst := 0;
		MesQInitial	:= MesDataExd.MesData.OUT_SetptQ ; 
	END_IF

	
	
TOF_FreqReg(IN:= MesDataExd.MesData.OUt_CmdFreqregMode, PT:= T#5S )  ; 	
	
FOR KK:= 1 TO ParamNbPcs DO 
MesDataExd.MesData.AX_PCS[KK].MesDeratingWord.4 := RS_VoltIsAbove.Q1 AND MesDataExd.MesData.OUT_CmdUregMode;
MesDataExd.MesData.AX_PCS[KK].MesDeratingWord.5 := RS_VoltIsBelow.Q1 AND MesDataExd.MesData.OUT_CmdUregMode;
MesDataExd.MesData.AX_PCS[KK].MesDeratingWord.6 := RS_FreqIsBelow.Q1 AND TOF_FreqReg.Q ;
MesDataExd.MesData.AX_PCS[KK].MesDeratingWord.7 := RS_FreqIsAbove.Q1 AND TOF_FreqReg.Q;
	
MesDataExd.MesData.AX_PCS[KK].MesDoorOpened := FALSE ; 
	
MesDataExd.MesData.MesOpeFlag.1 := MesDataExd.MesData.OUt_CmdFreqregMode; 
MesDataExd.MesData.MesOpeFlag.2 := MesDataExd.MesData.OUT_CmdUregMode ;

MesDataExd.MesData.MesOpeFlag.4 := MesDataExd.MesData.OUT_CmdQ; 
MesDataExd.MesData.MesOpeFlag.5 := MesDataExd.MesData.OUT_CmdCosPhi; 
MesDataExd.MesData.MesOpeFlag.6 :=  NOT MesDataExd.MesData.OUT_CmdGridMode; 
MesDataExd.MesData.MesOpeFlag.9 := TP_VoltRampToZeroOnceStable.Q OR TP_FreqRampToZeroSoClimit.Q OR TP_FreqRampToZeroOnceStable.Q  ; 
	
	
END_FOR
END_METHOD

METHOD M_Init

VAR 

END_VAR
SUPER^.M_Init() ; 

// 
MesData.OUT_CmdFreqRegMode := TRUE ; 
MesData.OUT_CmdURegMode := FALSE ;
END_METHOD

METHOD M_Read
//////////////////
//  Read Modbus Variable for PCS . 
/////////////////

VAR 
	// Method local variables (reinitialized at each cycle) 
	MW 						: FB_MergeWordsToDint; 

	
	MesPsetPt_Temp 			: REAL ;
	MesSetptQ_Temp			: REAL ;
	MesPavailablePcs_Temp	: REAL;
	MesPavailable_Temp		: REAL;
	
	ComErrorPcs_Temp		: WORD;
	
	KK						: BYTE;  					// FOR Loop 
	LL						: BYTE;						// Alarm Loop

	MesPsetPtPcs_temp		: ARRAY[1..CstNbPcs_Ess] OF  REAL; // Setpt lu sur le module
	MesSetptQPcs_temp		: ARRAY[1..CstNbPcs_Ess] OF  REAL;

	AX_Qty					: ARRAY[1..3] OF WORD := [68, 68, 68];
END_VAR
// Je récupère le clockRead et le.MesDataExd.MesData.(pour pouvoir réecrire les _Ack)
(*
ReadAds[2]
(
	NETID := '',
	PORT := ParamPort[3],
	IDXGRP := ParamGroup[3],
	IDXOFFS := ParamOffset[3],
	LEN := ParamLen[3],
	DESTADDR := ADR(ClockRead),
	READ := MAIN_Emul.MesWatchdog,
	TMOUT := T#100MS
);

ReadAds[4]		// Setpt P ANA
(
	NETID := '',
	PORT := ParamPort[6],
	IDXGRP := ParamGroup[6],
	IDXOFFS := ParamOffset[6],
	LEN := ParamLen[6],
	DESTADDR := ADR(OUt_SetptP_IO),
	READ := MAIN_Emul.MesWatchdog,
	TMOUT := T#100MS
);


ReadAds[6]		// Setpt Q ANA
(
	NETID := '',
	PORT := ParamPort[7],
	IDXGRP := ParamGroup[7],
	IDXOFFS := ParamOffset[7],
	LEN := ParamLen[7],
	DESTADDR := ADR(OUt_SetptQ_IO),
	READ := MAIN_Emul.MesWatchdog,
	TMOUT := T#100MS
);



ReadAds[5]
(
	NETID := '',
	PORT := ParamPort[2],
	IDXGRP := ParamGroup[2],
	IDXOFFS := ParamOffset[2],
	LEN := ParamLen[2],
	DESTADDR := ADR(MesDataExd.MesData.In),
	READ := MAIN_Emul.ClockReadIO,
	TMOUT := T#1S
);

Trig_ClockRead(CLK := ClockRead);

WriteAds[1]
(
	NETID := '',
	PORT := ParamPort[2],
	IDXGRP := ParamGroup[2],
	IDXOFFS := ParamOffset[2],
	LEN := ParamLen[2],
	SRCADDR := ADR(MesDataExd.MesData.,
	WRITE := Trig_ClockRead.Q AND NOT bTest,
	TMOUT := T#100MS
);
*)

// Je garde les tags calculés identiques
MesData.OUT_CmdP 						:= MesDataExd.MesData.In.out_CmdP					;

MesData.OUT_CmdBlackStart			:= MesDataExd.MesData.In.out_CmdBlackStart			;
MesData.OUT_CmdCosPhi               := MesDataExd.MesData.In.out_CmdCosPhi             ; 
MesData.OUT_CmdFreqregMode          := MesDataExd.MesData.In.out_CmdFreqregMode        ; 
MesData.OUT_CmdGridMode             := MesDataExd.MesData.In.out_CmdGridMode           ; 
MesData.OUT_CmdMicroCyclingMode     := MesDataExd.MesData.In.out_CmdMicroCyclingMode   ; 
MesData.OUT_CmdP                    := MesDataExd.MesData.In.out_CmdP                  ; 
MesData.OUT_CmdQ                    := MesDataExd.MesData.In.out_CmdQ                  ; 
MesData.OUT_CmdStandby              := MesDataExd.MesData.In.out_CmdStandby            ; 
MesData.OUT_CmdStop                 := MesDataExd.MesData.In.out_CmdStop               ; 
MesData.OUT_CmdStart                := MesDataExd.MesData.In.out_CmdStart              ; 
MesData.OUT_CmdUregMode             := MesDataExd.MesData.In.out_CmdUregMode           ; 
MesData.OUT_SetptCosPhi             := MesDataExd.MesData.In.out_SetptCosPhi           ; 
MesData.OUT_SetptP                  := MesDataExd.MesData.In.out_SetptP                ; 
MesData.OUT_SetptPMax               := MesDataExd.MesData.In.out_SetptPMax             ; 
MesData.OUT_SetptPMin               := MesDataExd.MesData.In.out_SetptPMin             ; 
MesData.OUT_SetptQ                  := MesDataExd.MesData.In.out_SetptQ                ; 
MesData.OUT_SetptQMax               := MesDataExd.MesData.In.out_SetptQMax             ; 
MesData.OUT_SetptQMin               := MesDataExd.MesData.In.out_SetptQMin             ; 
MesData.CalAlarm					:= MesDataExd.MesData.In.CalAlarm					;
MesData.CalAllAcClosed				:= MesDataExd.MesData.In.CalAllAcClosed			;	
MesData.CalAllDcClosed              := MesDataExd.MesData.In.CalAllDcClosed            ;  
MesData.CalAtLeastOneAcClosed       := MesDataExd.MesData.In.CalAtLeastOneAcClosed     ;  
MesData.CalAtLeastOneDcClosed       := MesDataExd.MesData.In.CalAtLeastOneDcClosed     ;  
MesData.CalAtLeastOnePcsConnected   := MesDataExd.MesData.In.CalAtLeastOnePcsConnected ;  
MesData.CalCosPhi                   := MesDataExd.MesData.In.CalCosPhi                 ;  
MesData.CalDynamicEfficiencyPcs     := MesDataExd.MesData.In.CalDynamicEfficiencyPcs   ;  
MesData.CalI                        := MesDataExd.MesData.In.CalI                      ;  
MesData.CalIdc                      := MesDataExd.MesData.In.CalIdc                    ;  
MesData.CalMaxS_ChargeFromBat       := MesDataExd.MesData.In.CalMaxS_ChargeFromBat     ;  
MesData.CalMaxS_DischargeFromBat    := MesDataExd.MesData.In.CalMaxS_DischargeFromBat  ;  
MesData.CalNbOnlinePcs              := MesDataExd.MesData.In.CalNbOnlinePcs            ;  
MesData.CalP                        := MesDataExd.MesData.In.CalP                      ;  
MesData.CalPdc                      := MesDataExd.MesData.In.CalPdc                    ;  
MesData.CalQ                        := MesDataExd.MesData.In.CalQ                      ;  
MesData.CalState                    := MesDataExd.MesData.In.CalState                  ;  
MesData.CalUac                      := MesDataExd.MesData.In.CalUac                    ;  
MesData.CalUdc                      := MesDataExd.MesData.In.CalUdc                    ;  
MesData.CalWarning                  := MesDataExd.MesData.In.CalWarning                ;  



ParamFreqRegSoCmax				:=  WORD_TO_REAL(AX_Cmd[1][2]	)	;
ParamFreqRegSoCmin				:=  WORD_TO_REAL(AX_Cmd[1][3]	)	;
MesSoCWrittenScada				:=  WORD_TO_REAL(AX_Cmd[1][4]	)	;
ParamQfU_UDbHigh			 	:=  WORD_TO_REAL(AX_Cmd[1][7] 	)	; 
ParamQfU_Umax				 	:=  WORD_TO_REAL(AX_Cmd[1][8] 	)	; 
ParamQfU_UDbLow				 	:=  WORD_TO_REAL(AX_Cmd[1][9] 	)	; 
ParamQfU_Umin				 	:=  WORD_TO_REAL(AX_Cmd[1][10] 	)	; 
ParamQfU_QDbHigh				:= -WORD_TO_REAL(AX_Cmd[1][11])*ParamPnomPcs/1000.0; 
ParamQfU_Qmax					:= -WORD_TO_REAL(AX_Cmd[1][12])*ParamPnomPcs/1000.0; 
ParamQfU_QDbLow					:= -WORD_TO_REAL(AX_Cmd[1][13])*ParamPnomPcs/1000.0; 
ParamQfU_Qmin					:= -WORD_TO_REAL(AX_Cmd[1][14])*ParamPnomPcs/1000.0; 
ParampfF_fDbHigh				:=  WORD_TO_REAL(AX_Cmd[1][21])/100.0;
ParamPfF_Fmax					:=  WORD_TO_REAL(AX_Cmd[1][22])/100.0;
ParamPfF_FDbLow					:=  WORD_TO_REAL(AX_Cmd[1][23])/100.0;
ParamPfF_Fmin					:=  WORD_TO_REAL(AX_Cmd[1][24])/100.0;
ParampfF_fDbHigh				:=  WORD_TO_REAL(AX_Cmd[1][25])/100.0;
ParamPfF_FDbLow					:=  WORD_TO_REAL(AX_Cmd[1][26])/100.0;
ParamPfF_FhystLow				:=  WORD_TO_REAL(AX_Cmd[1][27])/100.0;
ParamPfF_FhystHigh				:=  WORD_TO_REAL(AX_Cmd[1][28])/100.0;		
ParamPfF_PDbHigh				:=  INT_TO_REAL(WORD_TO_INT(AX_Cmd[1][29] ))*ParamPnom/1000.0; 
ParamPfF_Pmin					:=  INT_TO_REAL(WORD_TO_INT(AX_Cmd[1][30] ))*ParamPnom/1000.0; 
ParamPfF_PDbLow					:=  INT_TO_REAL(WORD_TO_INT(AX_Cmd[1][31] ))*ParamPnom/1000.0; 
ParamPfF_Pmax					:=  INT_TO_REAL(WORD_TO_INT(AX_Cmd[1][32] ))*ParamPnom/1000.0; 
ParamPfF_PDbHigh				:=  INT_TO_REAL(WORD_TO_INT(AX_Cmd[1][33] ))*ParamPnom/1000.0; 
ParamPfF_PDbLow					:=  INT_TO_REAL(WORD_TO_INT(AX_Cmd[1][34] ))*ParamPnom/1000.0; 
ParamTimeSoCRangeReachedRmp		:=	REAL_TO_TIME(REAL_TO_WORD(AX_Cmd[1][35]))*1000/10;				
ParamTimeEnterStblPriorRmp		:=	REAL_TO_TIME(REAL_TO_WORD(AX_Cmd[1][37]))*1000/10;					
ParamTimeFreqRegStbDuration		:=	REAL_TO_TIME(REAL_TO_WORD(AX_Cmd[1][36]))*1000/10;
END_METHOD

METHOD M_WriteCommand
//////////////////
//  Modbus Write of the command for the PCS. 
/////////////////

VAR 
	// Method local variables (reinitialized at each cycle) 
	
	AX_Adr			: ARRAY[1..5] OF UINT := [1707	, 1802	, 	0217 , 1735	,1741];
	AX_QTY			: ARRAY[1..5] OF BYTE := [28	, 33	, 	2	 , 6	,6];
	AX_UnitID		: ARRAY[1..5] OF BYTE := [1		, 1		, 	1	 , 1	,1];	

	KK: INT;



END_VAR
// Je récupère le clockWrite
(*
ReadAds[1]
(
	NETID := '',
	PORT := ParamPort[1],
	IDXGRP := ParamGroup[1],
	IDXOFFS := ParamOffset[1],
	LEN := ParamLen[1],
	DESTADDR := ADR(CmdWrite),
	READ := MAIN_Emul.MesWatchdog,
	TMOUT := T#100MS
);
*)
FOR KK := 1 TO 3 DO
	Trig_ClockWrite[KK](CLK := CmdWrite[KK]);
END_FOR
IF Trig_ClockWrite[1].Q THEN
	bTest := TRUE;
END_IF
(*
ReadADS[3]
(
	NETID := '',
	PORT := ParamPort[5],
	IDXGRP := ParamGroup[5],
	IDXOFFS := ParamOffset[5],
	LEN := ParamLen[5],
	DESTADDR := ADR(AX_CMD),
	READ := MAIN_Emul.MesWatchdog,
	TMOUT := T#100MS
);
*)
(*
FOR KK := 1 TO 3 DO
	IF Trig_ClockWrite[KK].Q THEN
		AX_CMD[KK] := AX_Cmd_New[KK];
	END_IF
END_FOR
*)
END_METHOD

END_FUNCTION_BLOCK

// ---- 01_Equipement_Library/ProtectRelay/FB_ProtectRelay_Base.TcPOU
FUNCTION_BLOCK FB_ProtectRelay_Base
//////////////////
// SEPAM system for High Voltage or Low Voltage Grid Protection. 
//////////////////
VAR_INPUT PERSISTENT
	// Parameters of the Object (instance/model specific) 
		ParamTempoComAlarm				: TIME := T#10S; 					// (s) Config : Tempo to detect LOC Alarm
		ParamTimeOut					: TIME := T#5S;						// (s) Modbus Timeout
		ParamClockReadTime				: TIME := T#2S;						// (s) Modbus Read Frequency
		ParamClockWriteTime				: TIME := T#1S;						// (s) Modbus Write Frequency



		ParamPTRNum							: UINT; // PTR Related to the Protect Relay 

END_VAR

VAR_INPUT 

	IN_CmdReset_L						: BOOL;			// (NA) External Reset Command	
    IN_CmdToggleRead					: BOOL;
    IN_CmdToggleWrite					: BOOL;
	                                    
	// I/O Inputs                       
		// GTE Protection LV            
		// WatchDog                     
	IN_MesWatchDog_IO					: BOOL:=TRUE;		// Watchdog is at True := Sepam OK
END_VAR

VAR_OUTPUT
	//Child objects
	
END_VAR

VAR
	Trig_ClockRead						: R_TRIG;
                                    	
	//M_ALARMMANAGEMENT VARIABLES// 	
                                    	                   
		TON_ComAlarm					: TON ; 												// Tempo before detecting loss of communication. 
	                                	
	//M_READ //                     	
		TP1								: TP;
		TP2								: TP;
		ClockRead		AT %Q*			: BOOL;
		ClockWrite						: BOOL;
		   		                    	
    //M_CP VARIABLES//              	
		Trig_Cmd_Read					: R_TRIG;                                                                                        
		Trig_Cmd_Write					: R_TRIG;                                                                                        
                                    	
		   		                    			
	//M_INIT VARIABLES // 	        			
		bInit							: BOOL := TRUE ; 		// (NA) Initialize object parameters at first cycle 
	
	
	// EMULATOR //
	

		
END_VAR

METHOD M_Execute
//////////////////
//  Method Calls 
/////////////////

VAR 
	// Method local variables (reinitialized at each cycle) 
	KK: UINT;
	MesStateCB : BOOL;
END_VAR
(*
Trig_ClockRead(CLK := ClockRead);


MesStateCB := A1_SUBMV.AX_FeederMVCB[ParamPTRNum].MesDataExd.MesData.MesClosed;
		
IF MesStateCB THEN
	MesData.MesI1 		:= AX_PTR[ParamPTRNum].MesDataExd.MesData.MesI ; 
	MesData.MesI2 		:= MesDataExd.MesData.MesI1 ; 
	MesData.MesI3 		:= MesDataExd.MesData.MesI1 ; 
	MesData.MesI0 		:= 0 ; 
ELSE            	
	MesData.MesI1 		:= 0 ;
	MesData.MesI2 		:= 0 ;
	MesData.MesI3 		:= 0 ;
	MesData.MesI0 		:= 0 ;
END_IF

MesData.MesImax1	:= MAX( MesDataExd.MesData.MesImax1, MesDataExd.MesData.MesI1) ; 
MesData.MesImax2	:= MAX( MesDataExd.MesData.MesImax2, MesDataExd.MesData.MesI2) ; 
MesData.MesImax3	:= MAX( MesDataExd.MesData.MesImax3, MesDataExd.MesData.MesI3) ; 
MesData.MesImax0	:= MAX( MesDataExd.MesData.MesImax0, MesDataExd.MesData.MesI0) ; 

//MesDataExd.MesData.MesClosed	        :=  MesStateCB ; 
//MesDataExd.MesData.MesOpened	        := NOT MesStateCB ; 
*)
END_METHOD

END_FUNCTION_BLOCK

// ---- 01_Equipement_Library/ProtectRelay/FB_ProtectRelay_DM2.TcPOU
FUNCTION_BLOCK FB_ProtectRelay_DM2 EXTENDS FB_ProtectRelay_Base
//////////////////
// REF615 + REU615 : communication not allowed by EDF 

VAR_OUTPUT
	//Child objects

END_VAR

VAR_INPUT
	IN_AlarmIMax_IO								: BOOL; //Max I Alarm, Losing autorisation and not possible to consumed
	IN_AlarmUmin_IO									: BOOL; //Min U , Keeping autorisation, If we have 3 gte in 30 min ==> Stop fedding and consumed during 2h
	IN_MesWatchdogREU615_IO						: BOOL:=TRUE ;// Watchdog . 0= alarm
	
END_VAR

VAR
	//M_ALARMMANAGEMENT VARIABLES//
	MesDataExd		: ProtectRelay_Standard ; 
	
	// EVALUATE //
	TON_GteIsLong	: TON ; 
	
	


		
END_VAR

METHOD M_AlarmManagement
//////////////////
// Manages Sepam Alarms. Alarms opens HT CB until Sepam manual Reset . Warning Opens CB-L but does not maintain warning
/////////////////

VAR 
	// Method local variables (reinitialized at each cycle) 
	FB_AlarmCodeManager 	: FB_AlarmCodeManager ; 

 
END_VAR


// ALARM CODE //
	FB_AlarmCodeManager(
		bAlarm1				:= MesDataExd.MesData.MesAlarmImax , 						// Max I>>0  fault 	 	
		bAlarm2				:= MesDataExd.MesData.MesAlarmUmin ,							// GTE fault 
		bAlarm3				:= MesDataExd.MesData.MesAlarmCom,						// Communication Alarm #COM
		bAlarm4				:= NOT IN_MesWatchDog_IO, 						// Watchdog REF615 not received      #COM 
		bAlarm5				:= NOT IN_MesWatchdogREU615_IO, 				// Watchdog REU615 not received	 #COM
		bAlarm6				:= FALSE, 									// 
		bAlarm7				:= FALSE, 									//
		bAlarm8				:= FALSE,                                   //
		bAlarm9				:= FALSE,                                   //
		bAlarm10			:= FALSE,                                   //
		bAlarm11			:= FALSE,                                   //
		bAlarm12			:= FALSE,                                   //
		bAlarm13			:= FALSE, 									//
		bAlarm14			:= FALSE, 									//
		bAlarm15			:= FALSE ,									// 
		wAlarmCode			=>MesDataExd.MesData.MesAlarmCode);

// WARNING CODE //
	FB_AlarmCodeManager(
		bAlarm1			:= FALSE , //
		bAlarm2			:= FALSE , //	
		bAlarm4			:= MesDataExd.MesData.MesAlarmUmin_Long, 						// GTE long 
		bAlarm5			:= FALSE, 									//
		bAlarm6			:= FALSE,                                   //
		bAlarm7			:= FALSE,                                   //
		bAlarm8			:= FALSE,                                   //
		bAlarm9			:= FALSE,                                   //
		bAlarm10		:= FALSE,                                   //
		bAlarm11		:= FALSE,                                   //
		bAlarm12		:= FALSE,                                   //
		bAlarm13		:= FALSE,                                   //
		bAlarm14		:= FALSE,                                   //
		bAlarm15		:= FALSE, 									//
		wAlarmCode		=>MesDataExd.MesData.MesWarningCode);

// EVENT CODE //
	FB_AlarmCodeManager(
		bAlarm1			:=FALSE, 		//  
		bAlarm2			:=FALSE, 		//  
		bAlarm3			:=FALSE, 		//  
		bAlarm4			:=FALSE, 		// 
		bAlarm5			:=FALSE,        //
		bAlarm6			:=FALSE,        //
		bAlarm7			:=FALSE,        //
		bAlarm8			:=FALSE,        //
		bAlarm9			:=FALSE,        //
		bAlarm10		:=FALSE,        //
		bAlarm11		:=FALSE,        //
		bAlarm12		:=FALSE,        //
		bAlarm13		:=FALSE,        //
		bAlarm14		:=FALSE,        //
		bAlarm15		:=FALSE, 
		wAlarmCode		=>MesDataExd.MesData.MesEventCode);
END_METHOD

METHOD M_Evaluate
VAR_INPUT
END_VAR
//Need to check the GTE FAULT


// GTE IS LONG AFTER 50S
TON_GteIsLong(IN:=IN_AlarmUmin_IO ,PT:=T#50S); 
MesData.MesAlarmUmin_Long := TON_GteIsLong.Q ; 


//Update MesData

MesData.MesAlarmUmin 			:= IN_AlarmUmin_IO;

TON_ComAlarm(IN:=NOT IN_MesWatchDog_IO OR NOT IN_MesWatchdogREU615_IO , PT:=ParamTempoComAlarm ) ; 
MesData.MesAlarmCom		:=TON_ComAlarm.Q  ; 
MesData.MesAlarmImax		:= IN_AlarmIMax_IO;
END_METHOD

END_FUNCTION_BLOCK

// ---- 01_Equipement_Library/ProtectRelay/FB_ProtectRelay_Flair23DM.TcPOU
FUNCTION_BLOCK FB_ProtectRelay_Flair23DM EXTENDS FB_ProtectRelay_Base
//////////////////
// SEPAM system for High Voltage or Low Voltage Grid Protection. 
//////////////////
VAR_INPUT PERSISTENT
	ParamTcpPort				: UINT:=502;                       // (NA) Tcp port 
	ParamIPAddress				: STRING; 						   // (NA) IP address
	ParamUnitID					: BYTE; 						   // (NA) Unit ID
END_VAR

VAR_INPUT 
	
END_VAR

VAR_OUTPUT
	
END_VAR

VAR_INPUT

END_VAR

VAR
MesDataExd	AT %Q*	: ProtectRelay_Flair23DM;     		//  MesDataExd.MesData.xd
	
	FB_ModbusRead	          	: ARRAY[1..3] OF FB_ModbusRead; 	// Modbus Read
									
	CalCP_Read					: BOOL;								
	CalCP_Write					: BOOL;
	
	MesBlock1_Temp 				: ARRAY [1..1] OF WORD ; 
	MesBlock2_Temp 				: ARRAY [1..15] OF WORD; 
	MesBlock3_Temp 				: ARRAY [1..2] OF WORD ; 
	
	AX_ModbusReadAlarm			: ARRAY[1..3] OF BOOL  ;
	AX_ModbusReadAlarmId		: ARRAY[1..3] OF UDINT ;	
	
	
	// EMIULATOR 
	Emul_AlarmCom			: BOOL ; // Flair CoM alarm 
	
	
END_VAR

METHOD M_Execute
//////////////////
//  Method Calls 
/////////////////

VAR 
	// Method local variables (reinitialized at each cycle) 
	MesU : REAL;
	MesV : REAL;
END_VAR
SUPER^.M_Execute() ; 

//COM
MesdataExd.MesStateCom 			:= Emul_AlarmCom;

// U
MesU := SEL(ABS(AX_PTR[ParamPTRNum].MesDataExd.MesData.MesI) < 0.001     , AX_PTR[ParamPTRNum].MesDataExd.MesData.MesP/AX_PTR[ParamPTRNum].MesDataExd.MesData.MesI , 0);

MesDataExd.MesData.MesU12	:= MesU;
MesDataExd.MesData.MesU23	:= MesU;
MesDataExd.MesData.MesU31	:= MesU;
                            
// V                        
MesDataExd.MesV1			:= MesU/SQRT(3); 
MesDataExd.MesV2			:= MesU/SQRT(3); 
MesDataExd.MesV3			:= MesU/SQRT(3); 
MesDataExd.MesV0			:= 0;
END_METHOD

END_FUNCTION_BLOCK

// ---- 01_Equipement_Library/ProtectRelay/FB_ProtectRelay_NSXCB.TcPOU
FUNCTION_BLOCK FB_ProtectRelay_NSXCB EXTENDS FB_ProtectRelay_Base
//////////////////
// SEPAM system for High Voltage or Low Voltage Grid Protection. 
//////////////////
VAR_INPUT PERSISTENT
	ParamTcpPort				: UINT:=502;		// (NA) Tcp port 
	ParamIPAddress				: STRING;           // (NA) IP address
	ParamUnitID					: BYTE;             // (NA) Unit ID
END_VAR

VAR_INPUT 

END_VAR

VAR_OUTPUT
	
END_VAR

VAR_INPUT

END_VAR

VAR
MesDataExd	AT %Q*	: ProtectRelay_NSXCB;
	
	FB_ModbusRead	          	: ARRAY[1..3] OF FB_ModbusRead; 
		
	CalCP_Read					: BOOL;
	CalCP_Write                 : BOOL;
	
	MesBlock1_Temp 				: ARRAY [1..1] OF WORD ; 
	MesBlock2_Temp 				: ARRAY [1..32] OF WORD ; 
	MesBlock3_Temp 				: ARRAY [1..8] OF WORD ; 
	
	AX_ModbusReadAlarm			: ARRAY[1..3] OF BOOL;
	AX_ModbusReadAlarmId		: ARRAY[1..3] OF UDINT;	
	
	// Emulator
	Emul_StateCom : BOOL := FALSE;
END_VAR

METHOD M_Execute
//////////////////
//  Method Calls 
/////////////////

VAR 
	// Method local variables (reinitialized at each cycle) 
KK : INT;

END_VAR
SUPER^.M_Execute(); 

//COM
MesdataExd.MesStatCom  := Emul_StateCom;
            
///MesDataExd.MesData.MesPtot := // AX_PTR[ParamPTRNum].MesDataExd.MesData.MesP;
     
MesdataExd.MesP1 := AX_PTR[ParamPTRNum].MesDataExd.MesData.MesP;   
MesdataExd.MesP2 := MesDataExd.MesData.MesP1;	 	
MesdataExd.MesP3 := MesDataExd.MesData.MesP1;	 	
               
MesdataExd.MesQ1 := AX_PTR[ParamPTRNum].MesDataExd.MesData.MesQ; 	 	
MesdataExd.MesQ2 := MesDataExd.MesData.MesQ1;	 	
MesdataExd.MesQ3 := MesDataExd.MesData.MesQ1; 	

// S 	         
MesdataExd.MesS1 :=  SQRT( MesDataExd.MesData.MesP1*.MesDataExd.MesData.MesP1 + MesDataExd.MesData.MesQ1.MesDataExd.MesData.MesQ1) ;
MesdataExd.MesS2 := MesDataExd.MesData.MesS1; 	
MesdataExd.MesS3 := MesDataExd.MesData.MesS1;	
MesdataExd.MesStot := SQRT( MesDataExd.MesData.MesPtot * MesDataExd.MesData.MesPtot + MesDataExd.MesData.MesQtot.MesDataExd.MesData.MesQtot);	 
	                  

IF MesDataExd.MesData.MesPtot > 0 THEN
MesDataExd.MesData.MesEact := MesDataExd.MesData.MesEact + MesDataExd.MesData.MesPtot*ParamCycleTime_Emul/3600000	; // Ptot ? 
END_IF

IF MesDataExd.MesData.MesQtot > 0 THEN
MesDataExd.MesData.MesEReact := MesDataExd.MesData.MesEReact + MesDataExd.MesData.MesQtot*ParamCycleTime_Emul/3600000	; // Qtot ? 
END_IF

MesdataExd.MesCosPhi  := MesDataExd.MesData.MesPtot.MesDataExd.MesData.MesStot;	                  
MesdataExd.MesCosPhi1 := MesDataExd.MesData.MesCosPhi;
MesdataExd.MesCosPhi2 := MesDataExd.MesData.MesCosPhi;
MesdataExd.MesCosPhi3 := MesDataExd.MesData.MesCosPhi;
	
Mesdata.MesFreq := A1_SUBMV.MesDataExd.MesData.MesFreq;
MesdataExd.MesMaxFreq := 52;
END_METHOD

END_FUNCTION_BLOCK

// ---- 01_Equipement_Library/ProtectRelay/FB_ProtectRelay_PACE100ST.TcPOU
FUNCTION_BLOCK FB_ProtectRelay_PACE100ST EXTENDS FB_ProtectRelay_Base
//////////////////
// SEPAM system for High Voltage or Low Voltage Grid Protection . 
//////////////////


VAR_INPUT PERSISTENT
	// Parameters of the Object (instance/model specific) 
	ParamInInterfaceSub						: BOOL := TRUE; // Serial interface RS422/RS485 TYPE (0:EL6021,1:SUB9)
END_VAR

VAR_OUTPUT

END_VAR

VAR_INPUT
	InUnitID            					: DINT;			// (NA)   ID FOR SEPAM S48 Modbus Unit ID. 	

	IN_MesAlarmI0Max_IO								: BOOL;
	IN_MesAlarmIMax_IO								: BOOL;
END_VAR

VAR

	ModbusRTU								: FB_ModbusRTU;
	MesBlock								: ARRAY[1..3] OF ARRAY[1..120] OF WORD;	
	AX_Addr									: ARRAY[1..3] OF UINT 	:= [1200,	1500,	2000];
	AX_Qty									: ARRAY[1..3] OF UINT	:= [2,		2,		3];
	AX_UnitId								: ARRAY[1..3] OF BYTE	:= [1,		1,		1];
	AX_Function								: ARRAY[1..3] OF UINT	:= [4,		4,		4];	
	AX_Priority								: ARRAY[1..3] OF UINT	:= [1,		1,		1];
	AX_bStart								: ARRAY[1..3] OF BOOL;
	AX_TrigRead								: ARRAY[1..3] OF R_trig;
	MbStruct								: ARRAY[1..3] OF Struct_InputRTU;	
	
	KK										: INT;

MesDataExd				AT %Q* 	: ProtectRelay_PACE100ST ;
	
	//M_EVALUATE

	//ClockRead								: BOOL;

END_VAR

METHOD M_AlarmManagement
//////////////////
// Manages Sepam Alarms. Alarms opens HT CB until Sepam manual Reset . Warning Opens CB-L but does not maintain warning
/////////////////

VAR 
	// Method local variables (reinitialized at each cycle) 
	FB_AlarmCodeManager 	: FB_AlarmCodeManager ; 

END_VAR

// ALARM CODE //
	FB_AlarmCodeManager(
		bAlarm1				:= MesDataExd.MesData.CB_In_Alarm,		// CB in Alarm
		bAlarm2				:= IN_MesAlarmI0Max_IO,					// Max IO Fault
		bAlarm3				:= IN_MesAlarmIMax_IO,						// Max I Fault 
		bAlarm4				:= FALSE,						// 
		bAlarm5				:= FALSE,						//
		bAlarm6				:= FALSE, 						// 
		bAlarm7				:= FALSE, 						// 
		bAlarm8				:= FALSE, 						// 
		bAlarm9				:= FALSE, 						// 
		bAlarm10			:= FALSE, 						// 
		bAlarm11			:= FALSE, 						//
		bAlarm12			:= FALSE, 						// 
		bAlarm13			:= FALSE, 						//
		bAlarm14			:= FALSE, 						//
		bAlarm15			:= FALSE, 						// 
		wAlarmCode			=>MesDataExd.MesData.MesAlarmCode);

// WARNING CODE //
	FB_AlarmCodeManager(
		bAlarm1			:= FALSE,//
		bAlarm2			:= FALSE,//
		bAlarm4			:= FALSE,//
		bAlarm5			:= FALSE,//
		bAlarm6			:= FALSE,// 
		bAlarm7			:= FALSE,// 
		bAlarm8			:= FALSE,// 
		bAlarm9			:= FALSE,// 
		bAlarm10		:= FALSE,// 
		bAlarm11		:= FALSE,// 
		bAlarm12		:= FALSE,// 
		bAlarm13		:= FALSE,// 
		bAlarm14		:= FALSE,// 
		bAlarm15		:= FALSE,// 
		wAlarmCode		=>MesDataExd.MesData.MesWarningCode);

// EVENT CODE //
	FB_AlarmCodeManager(
		bAlarm1			:=FALSE, 		// 
		bAlarm2			:=FALSE, 		// 
		bAlarm3			:=FALSE, 		// 
		bAlarm4			:=FALSE, 		// 
		bAlarm5			:=FALSE, 		//
		bAlarm6			:=FALSE, 		//
		bAlarm7			:=FALSE, 		//
		bAlarm8			:=FALSE, 		//
		bAlarm9			:=FALSE, 		//
		bAlarm10		:=FALSE, 		//
		bAlarm11		:=FALSE, 		//
		bAlarm12		:=FALSE, 		//
		bAlarm13		:=FALSE, 		//
		bAlarm14		:=FALSE, 		//
		bAlarm15		:=FALSE, 		//
		wAlarmCode		=>MesDataExd.MesData.MesEventCode);
END_METHOD

METHOD M_Evaluate
VAR_INPUT
END_VAR

VAR
	CloseMainMVCB							: BOOL;
	Valtemp									: REAL;
	MesConnectAuthorization					: BOOL;

END_VAR
END_METHOD

METHOD M_Init
VAR_INPUT
END_VAR
//Modbus RTU Relay
FOR KK := 1 TO 4 DO 
	MbStruct[KK].InBuffer := ADR(MesBlock[KK]);
	MbStruct[KK].InFunction := AX_Function[KK];
	MbStruct[KK].InQuantity := AX_Qty[KK];
	MbStruct[KK].InStartAddr := AX_Addr[KK];
	MbStruct[KK].InUnitID := AX_UnitId[KK];
END_FOR
END_METHOD

METHOD M_Read
//////////////////
//  Method Calls 
/////////////////

VAR 
//local variables (reinitialized at each cycle) 
	MW 					: FB_MergeWordsToDint; 
	MW_Float			: FB_MergeWordsToFloat; 
END_VAR

MesDataExd.MesData.= MesDataExd.MesData.;

IF MesCP_Read THEN	

ModbusRTU();


FOR KK := 1 TO 4 DO
	AX_TrigRead[KK](CLK  :=CalLocalTimeStruct.wSecond MOD 5 = 0);
	IF AX_TrigRead[KK].Q THEN
		ModbusRTU.M_AddAction_FIFO(InStruct := MbStruct[KK], InPriority := AX_Priority[KK]);
	END_IF
END_FOR


MW_Float( WORD_STRONG_F:= MesBlock[1][1], 	WORD_WEAK_F := MesBlock[1][2],  NUMBER_F:= MesDataExd.MesData.MesI1);
MW_Float( WORD_STRONG_F:= MesBlock[1][3], 	WORD_WEAK_F := MesBlock[1][4],  NUMBER_F:= MesDataExd.MesData.MesI2);
MW_Float( WORD_STRONG_F:= MesBlock[1][5], 	WORD_WEAK_F := MesBlock[1][6],  NUMBER_F:= MesDataExd.MesData.MesI3);
MW_Float( WORD_STRONG_F:= MesBlock[1][7], 	WORD_WEAK_F := MesBlock[1][8],  NUMBER_F:= MesDataExd.MesData.MesI0);
MW_Float( WORD_STRONG_F:= MesBlock[1][15], 	WORD_WEAK_F := MesBlock[1][16], NUMBER_F:= MesDataExd.MesData.Thermal_Overload);
MW_Float( WORD_STRONG_F:= MesBlock[1][17], 	WORD_WEAK_F := MesBlock[1][18], NUMBER_F:= MesDataExd.MesData.MesFreq);


MesDataExd.Comut 			:= WORD_TO_BOOL(MesBlock[2][7]);
MesDataExd.CB_Close 		:= WORD_TO_BOOL(MesBlock[2][8]);
MesDataExd.CB_In_Alarm 		:= WORD_TO_BOOL(MesBlock[2][9]);
MesDataExd.Trip_Counter 	:= WORD_TO_INT(MesBlock[3][3]);

END_IF
END_METHOD

END_FUNCTION_BLOCK

// ---- 01_Equipement_Library/ProtectRelay/FB_ProtectRelay_REF615.TcPOU
FUNCTION_BLOCK FB_ProtectRelay_REF615 EXTENDS FB_ProtectRelay_Base
VAR_INPUT PERSISTENT
		ParamIPAddress				: STRING 	:= '192.168.20.66'; 	// (NA)Config: IP Adress of PV INverter
		ParamUnitID 				: BYTE  	:= 1; 			  		// (NA)   Modbus Unit ID. 
		ParamTCPPort				: UINT		:= 502;					// (NA) TCP port for modbus
		

//		ParamTempoComAlarm			: TIME 		:= T#2S;
//		ParamTempoComWarning		: TIME		:= T#2S;
		ParamNominalCurrent			: REAL 		:= 100 ; 				// (A) Nominal current set in the protection relay.
		
END_VAR

VAR
	// M_ALARMMANAGEMENT		
//		TON_ComAlarm				: TON;
//		TON_ComWarning				: TON;	
//		MesWarningCom				: BOOL;
//		MesAlarmCom					: BOOL;
	// M_READ VARIABLES//
		AX_ModbusRead		   		: ARRAY [1..3] OF FB_ModbusRead ; 					// (NA) FB for Modbus Reading
		                                        
		MesBlock_Temp 				: ARRAY [1..3] OF ARRAY[1..120]  OF WORD; 			// (NA) Temporary Block with multiple modbus reading (Caution : Double Word variables)

	MesDataExd		AT %Q* 	: ProtectRelay_REFIO ; 
	

	// M_STATEMANAGER//
	
END_VAR

METHOD M_AlarmManagement
//////////////////
// Manages IntelliGen Alarms
/////////////////

VAR 
	// Method local variables (reinitialized at each cycle) 
	FB_AlarmCodeManager : FB_AlarmCodeManager ; 

	KK					: BYTE;		// For Loop 
	
	ComWarning			: BOOL;		// Aggregated Wcommunication warning
	ComAlarm			: BOOL;		// Aggregated communication Alarm

	MesWarningCom: BOOL;
END_VAR

	//Alarm
	
	TON_ComAlarm	(IN:= (AX_ModbusRead[1].ModbusReadAlarm) AND (AX_ModbusRead[2].ModbusReadAlarm) AND (AX_ModbusRead[3].ModbusReadAlarm) , PT:= ParamTempoComAlarm, 	Q= MesDataExd.MesData.MesAlarmCom) ;	
//	TON_ComWarning	(IN:= (AX_ModbusRead[1].ModbusReadAlarm) OR  (AX_ModbusRead[2].ModbusReadAlarm) OR  (AX_ModbusRead[3].ModbusReadAlarm) , PT:= ParamTempoComWarning, 	Q=>MesWarningCom) ;	

	MesWarningCom :=(AX_ModbusRead[1].ModbusReadAlarm) OR  (AX_ModbusRead[2].ModbusReadAlarm) OR  (AX_ModbusRead[3].ModbusReadAlarm) ; 


	
// ALARM CODE //
	FB_AlarmCodeManager(
		bAlarm1			:= MesDataExd.MesData.MesAlarmImax,  				//  Max I>>0  fault  
		bAlarm2			:= FALSE , 										//
		bAlarm3			:= MesDataExd.MesData.MesAlarmCom , 			// Communication alarm #COM
		bAlarm4			:= MesDataExd.MesData.MesAlarmTCS, 		        // Trip circuit Supervision alarm .     
		bAlarm5			:= FALSE, 										// 
		bAlarm6			:= FALSE, 										// 
		bAlarm7			:= False, 										// 
		bAlarm8			:= False, 										// 
		bAlarm9			:= FALSE, 										//
		bAlarm10		:= FALSE, 										//
		bAlarm11		:= FALSE,                       				//
		bAlarm12		:= FALSE,                       				//
		bAlarm13		:= FALSE, 										//
		bAlarm14		:= FALSE, 										// 
		bAlarm15		:= FALSE , 										// 
		wAlarmCode		=>MesDataExd.MesData.MesAlarmCode);

// WARNING CODE //
	FB_AlarmCodeManager(
 		bAlarm1			:= MesWarningCom,								// Bad communication	#COM			
		bAlarm2			:= FALSE ,										// 
		bAlarm3			:= FALSE , 										//		
		bAlarm4			:= FALSE, 						                //
		bAlarm5			:= FALSE, 						                //
		bAlarm6			:= FALSE, 						                //
		bAlarm7			:= FALSE,                                       //
		bAlarm8			:= FALSE,                                       //
		bAlarm9			:= FALSE,                                       //
		bAlarm10		:= FALSE,                                       //
		bAlarm11		:= FALSE,                                       //
		bAlarm12		:= FALSE,                                       //
		bAlarm13		:= FALSE,                                       //
		bAlarm14		:= FALSE,                                       //
		bAlarm15		:= FALSE,                                       //
		wAlarmCode		=>MesDataExd.MesData.MesWarningCode);	

// EVENT CODE //
	FB_AlarmCodeManager(
 		bAlarm1			:= FALSE,		//				
		bAlarm2			:= FALSE,	    //
		bAlarm3			:= FALSE,		//	
		bAlarm4			:= FALSE, 		//				
		bAlarm5			:= FALSE, 		//				
		bAlarm6			:= FALSE, 		//				
		bAlarm7			:= FALSE,       //
		bAlarm8			:= FALSE,       //
		bAlarm9			:= FALSE,       //
		bAlarm10		:= FALSE,       //
		bAlarm11		:= FALSE,       //
		bAlarm12		:= FALSE,       //
		bAlarm13		:= FALSE,       //
		bAlarm14		:= FALSE,       //
		bAlarm15		:= FALSE,       //
		wAlarmCode		=>MesDataExd.MesData.MesEventCode);
END_METHOD

METHOD M_Read
//////////////////
//  Read Modbus Variable for PCS . 
/////////////////
VAR 
	// Method local variables (reinitialized at each cycle) 
		
		AX_Addr				: ARRAY[1..3] OF UINT := [138, 		9409, 	171 ];
		AX_Qty				: ARRAY[1..3] OF UINT := [4, 		4, 	36	];
		
	
END_VAR


IF MesCP_Read THEN	
MesDataExd.MesData.:= MesDataExd.MesData.; // Allow to initialize.MesDataExd.MesData.with code from RPN_Base ; 

AX_ModbusRead[1]
(
	pDestAddr 		:= ADR(MesBlock_Temp[1]),
	sIPAddr 		:= ParamIPAddress,
	tTimeout 		:= ParamTimeout,
	nQuantity 		:= AX_Qty[1],
	ntcpport 		:= ParamTCPPort,
	nMBAddr 		:= AX_Addr[1]-1,
	nUnitID 		:= ParamUnitID,
	cbLength 		:= SIZEOF(MesBlock_Temp[1]),
	ClockRead 		:= ClockRead AND MesCP_Read,
	Reset 			:= CmdClearFault_G OR IN_CmdReset_L,
);

AX_ModbusRead[2]
(
	pDestAddr 		:= ADR(MesBlock_Temp[2]),
	sIPAddr 		:= ParamIPAddress,
	tTimeout 		:= ParamTimeout,
	nQuantity 		:= AX_Qty[2],
	ntcpport 		:= ParamTCPPort,
	nMBAddr 		:= AX_Addr[2]-1,
	nUnitID 		:= ParamUnitID,
	cbLength 		:= SIZEOF(MesBlock_Temp[2]),
	ClockRead 		:= ClockRead AND MesCP_Read,
	Reset 			:= CmdClearFault_G OR IN_CmdReset_L
);

AX_ModbusRead[3]
(
	pDestAddr 		:= ADR(MesBlock_Temp[3]),
	sIPAddr 		:= ParamIPAddress,
	tTimeout 		:= ParamTimeout,
	nQuantity 		:= AX_Qty[3],
	ntcpport 		:= ParamTCPPort,
	nMBAddr 		:= AX_Addr[3]-1,
	nUnitID 		:= ParamUnitID,
	cbLength 		:= SIZEOF(MesBlock_Temp[3]),
	ClockRead 		:= ClockRead AND MesCP_Read,
	Reset 			:= CmdClearFault_G OR IN_CmdReset_L
);



	


MesDataExd.MesData.MesI1 	:= WORD_TO_REAL(MesBlock_Temp[1][1])/1000*ParamNominalCurrent;
MesDataExd.MesData.MesI2 	:= WORD_TO_REAL(MesBlock_Temp[1][2])/1000*ParamNominalCurrent;
MesDataExd.MesData.MesI3 	:= WORD_TO_REAL(MesBlock_Temp[1][3])/1000*ParamNominalCurrent;
MesDataExd.MesData.MesI0 	:= WORD_TO_REAL(MesBlock_Temp[1][4])/1000*ParamNominalCurrent;


MesDataExd.MesData.MesImax1	:= WORD_TO_REAL(MesBlock_Temp[2][1])/1000*ParamNominalCurrent;
MesDataExd.MesData.MesImax2	:= WORD_TO_REAL(MesBlock_Temp[2][2])/1000*ParamNominalCurrent;
MesDataExd.MesData.MesImax3	:= WORD_TO_REAL(MesBlock_Temp[2][3])/1000*ParamNominalCurrent;
MesDataExd.MesData.MesImax0	:= WORD_TO_REAL(MesBlock_Temp[2][4])/1000*ParamNominalCurrent;


MesDataExd.MesTransfoAlarm		:= MesBlock_Temp[3][31].0 ;
MesDataExd.MesSWOpened			:= MesBlock_Temp[3][31].4 ;
MesDataExd.MesSWClosed			:= MesBlock_Temp[3][31].6 ;
MesDataExd.MesEarth				:= MesBlock_Temp[3][31].8 ;
MesDataExd.MesSF6Low			:= MesBlock_Temp[3][31].10;
MesDataExd.MesSF6Unsufficient	:= MesBlock_Temp[3][31].12;
MesDataExd.MesTransfoWarning		:= MesBlock_Temp[3][31].14;

MesDataExd.MesClosed	        := MesBlock_Temp[3][30].2;
MesDataExd.MesOpened	        := MesBlock_Temp[3][30].4;
MesDataExd.MesComutLocal				:= NOT MesBlock_Temp[3][30].6;

MesDataExd.MesData.MesAlarmImax				:= MesBlock_Temp[3][3].1 ; // Max I ou Max I Inverse. Maintenu jusque l'acquittement.  
//MesDataExd.MesData.MesAlarmTCS				:=  ; 

END_IF

//MesDataExd.MesData.MesAlarmUminrmUmin	:= ; 

// Properties update
MesDataExd.MesData.MesI := MesDataExd.MesData.MesI1 + MesDataExd.MesData.MesI2 + MesDataExd.MesData.MesI3)/3 ;
END_METHOD

END_FUNCTION_BLOCK

// ---- 01_Equipement_Library/ProtectRelay/FB_ProtectRelay_SEPAM10a.TcPOU
FUNCTION_BLOCK FB_ProtectRelay_SEPAM10a EXTENDS FB_ProtectRelay_Base
VAR_INPUT
	InUnitID            : DINT;			// (NA)   SMA Modbus Unit ID. 
	
END_VAR
VAR_OUTPUT
	OutFBCompleteted   : BOOL;
	
END_VAR
VAR
// M_ALARMMNGMT VARIABLES //
		MesAlarmCode				: WORD ;  			// (NA) [P,H,B]   Alarm Word . 0: Synthesis , 1:SMA general alarm , 2:Communication Alarm , 3:, 4:, 5:, 6:, 7:, 8:, 9:, 10:, 11:, 12:, 13:, 14:, 15:, 16:
		MesWarningCode				: WORD ;  			// (NA) [P,H,B]   Warning Word . 0: Synthesis , 1:SMA general warning  , 2: , 3: , 4:, 5:, 6:, 7:, 8:, 9:, 10:, 11:, 12:, 13:, 14:, 15:, 16:		
  		MesEventCode				: WORD; 			// (NA) [P,H,B] Event Code. Acknowledgable.
                                              		

		MesComError					: BOOL ; 			// (NA) [P,H]  True if lost of communication
		MesAlarmCom					: BOOL ; 			// (NA) All modbus trame fail 
		
	// M_READ VARIABLES//
		FB_ModbusRead_I1          	: FB_ReadModbusRTU_V2; 				// (NA) FB for Modbus Reading
		MesDataExd		      	AT %Q* 	: ProtectRelay_S48; 	
		MesBlock1_Temp 				: ARRAY[0..7]  OF WORD; 			// (NA) Temporary Block with multiple modbus reading (Caution : Double Word variables)
		AX_bRead 					: ARRAY[1..2]  OF BOOL;
		ModbusReadAlarm             : BOOL;				// (NA) Modbus Read Alarm for communications
		MesModbusAlarmCode			: UDINT;							// (NA) Modbus Read Alarm Code
		CalAllCompleted				: BOOL;								// (NA) Returns the status of all modbus requests
	
		AllNotBusy					: BOOL:=TRUE;
		TP_Read						: LTP; 								// (NA) Tempo to define Modbus Reading Frequency
	//	ClockRead					: BOOL;								// (NA) Modbus reading Clock
		RTrig						: R_TRIG;
END_VAR

